LIN {X 0,Y 312.688,Z 380.055,A -85,B 0,C 180,E1 -15702.753,E2 -15702.753} C_VEL
LIN {X 0,Y 311.794,Z 385.413,A -85,B 0,C 180,E1 -15704.959,E2 -15704.959} C_VEL
LIN {X 0,Y 311.134,Z 389.57,A -85,B 0,C 180,E1 -15707.342,E2 -15707.342} C_VEL
LIN {X 0,Y 310.753,Z 391.625,A -85,B 0,C 180,E1 -15709.017,E2 -15709.017} C_VEL
LIN {X 0,Y 310.505,Z 392.931,A -85,B 0,C 180,E1 -15710.675,E2 -15710.675} C_VEL
LIN {X 0,Y 310.399,Z 393.625,A -85,B 0,C 180,E1 -15712.415,E2 -15712.415} C_VEL
LIN {X 0,Y 310.321,Z 393.447,A -85,B 0,C 180,E1 -15714.617,E2 -15714.617} C_VEL
LIN {X 0,Y 310.452,Z 391.861,A -85,B 0,C 180,E1 -15717.093,E2 -15717.093} C_VEL
LIN {X 0,Y 310.763,Z 389.249,A -85,B 0,C 180,E1 -15719.246,E2 -15719.246} C_VEL
LIN {X 0,Y 311.221,Z 384.676,A -85,B 0,C 180,E1 -15721.725,E2 -15721.725} C_VEL
LIN {X 0,Y 311.824,Z 379.437,A -85,B 0,C 180,E1 -15723.802,E2 -15723.802} C_VEL
LIN {X 0,Y 312.576,Z 373.086,A -85,B 0,C 180,E1 -15725.776,E2 -15725.776} C_VEL
LIN {X 0,Y 313.482,Z 365.782,A -85,B 0,C 180,E1 -15727.598,E2 -15727.598} C_VEL
LIN {X 0,Y 314.661,Z 356.752,A -85,B 0,C 180,E1 -15729.403,E2 -15729.403} C_VEL
LIN {X 0,Y 315.916,Z 346.753,A -85,B 0,C 180,E1 -15731.015,E2 -15731.015} C_VEL
LIN {X 0,Y 317.246,Z 335.532,A -85,B 0,C 180,E1 -15732.453,E2 -15732.453} C_VEL
LIN {X 0,Y 318.469,Z 323.461,A -85,B 0,C 180,E1 -15733.66,E2 -15733.66} C_VEL
LIN {X 0,Y 319.474,Z 310.963,A -85,B 0,C 180,E1 -15734.613,E2 -15734.613} C_VEL
LIN {X 0,Y 320.299,Z 298.124,A -85,B 0,C 180,E1 -15735.304,E2 -15735.304} C_VEL
LIN {X 0,Y 320.899,Z 284.464,A -85,B 0,C 180,E1 -15735.77,E2 -15735.77} C_VEL
LIN {X 0,Y 322.484,Z 214.178,A -85,B 0,C 180,E1 -15737.436,E2 -15737.436} C_VEL
LIN {X 0,Y 318.5,Z 192.839,A -85,B 0,C 180,E1 -15738.248,E2 -15738.248} C_VEL
LIN {X 0,Y 315.024,Z 182.877,A -85,B 0,C 180,E1 -15738.777,E2 -15738.777} C_VEL
LIN {X 0,Y 314.543,Z 180.395,A -85,B 0,C 180,E1 -15739.453,E2 -15739.453} C_VEL
LIN {X 0,Y 312.923,Z 171.315,A -85,B 0,C 180,E1 -15742.419,E2 -15742.419} C_VEL
LIN {X 0,Y 312.873,Z 171.01,A -85,B 0,C 180,E1 -15742.905,E2 -15742.905} C_VEL
LIN {X 0,Y 312.933,Z 171.005,A -85,B 0,C 180,E1 -15747.427,E2 -15747.427} C_VEL
LIN {X 0,Y 313.099,Z 170.983,A -85,B 0,C 180,E1 -15750.001,E2 -15750.001} C_VEL
LIN {X 0,Y 312.934,Z 171.002,A -85,B 0,C 180,E1 -15752.576,E2 -15752.576} C_VEL
LIN {X 0,Y 312.89,Z 171.008,A -85,B 0,C 180,E1 -15756.45,E2 -15756.45} C_VEL
LIN {X 0,Y 312.684,Z 171.033,A -85,B 0,C 180,E1 -15760.36,E2 -15760.36} C_VEL
LIN {X 0,Y 312.699,Z 171.032,A -85,B 0,C 180,E1 -15764.889,E2 -15764.889} C_VEL
LIN {X 0,Y 312.63,Z 171.041,A -85,B 0,C 180,E1 -15769.238,E2 -15769.238} C_VEL
LIN {X 0,Y 312.545,Z 171.052,A -85,B 0,C 180,E1 -15772.79,E2 -15772.79} C_VEL
LIN {X 0,Y 312.596,Z 171.039,A -85,B 0,C 180,E1 -15775.934,E2 -15775.934} C_VEL
LIN {X 0,Y 312.538,Z 171.052,A -85,B 0,C 180,E1 -15779.652,E2 -15779.652} C_VEL
LIN {X 0,Y 312.519,Z 171.052,A -85,B 0,C 180,E1 -15783.69,E2 -15783.69} C_VEL
LIN {X 0,Y 312.52,Z 171.051,A -85,B 0,C 180,E1 -15787.387,E2 -15787.387} C_VEL
LIN {X 0,Y 312.49,Z 171.06,A -85,B 0,C 180,E1 -15790.71,E2 -15790.71} C_VEL
LIN {X 0,Y 312.473,Z 171.059,A -85,B 0,C 180,E1 -15794.207,E2 -15794.207} C_VEL
LIN {X 0,Y 312.447,Z 171.057,A -85,B 0,C 180,E1 -15795.292,E2 -15795.292} C_VEL
LIN {X 0,Y 311.803,Z 171.141,A -85,B 0,C 180,E1 -15796.368,E2 -15796.368} C_VEL
LIN {X 0,Y 308.949,Z 171.49,A -85,B 0,C 180,E1 -15798.119,E2 -15798.119} C_VEL
LIN {X 0,Y 306.523,Z 171.792,A -85,B 0,C 180,E1 -15799.54,E2 -15799.54} C_VEL
LIN {X 0,Y 305.494,Z 171.926,A -85,B 0,C 180,E1 -15800.64,E2 -15800.64} C_VEL
LIN {X 0,Y 305.417,Z 171.93,A -85,B 0,C 180,E1 -15801.012,E2 -15801.012} C_VEL
LIN {X 0,Y 305.462,Z 171.935,A -85,B 0,C 180,E1 -15804.888,E2 -15804.888} C_VEL
LIN {X 0,Y 305.442,Z 171.938,A -85,B 0,C 180,E1 -15808.359,E2 -15808.359} C_VEL
LIN {X 0,Y 305.477,Z 171.931,A -85,B 0,C 180,E1 -15811.11,E2 -15811.11} C_VEL
LIN {X 0,Y 305.502,Z 171.93,A -85,B 0,C 180,E1 -15814.082,E2 -15814.082} C_VEL
LIN {X 0,Y 305.484,Z 171.933,A -85,B 0,C 180,E1 -15818.402,E2 -15818.402} C_VEL
LIN {X 0,Y 305.591,Z 171.916,A -85,B 0,C 180,E1 -15821.218,E2 -15821.218} C_VEL
LIN {X 0,Y 305.651,Z 171.906,A -85,B 0,C 180,E1 -15825.35,E2 -15825.35} C_VEL
LIN {X 0,Y 305.626,Z 171.913,A -85,B 0,C 180,E1 -15829.4,E2 -15829.4} C_VEL
LIN {X 0,Y 305.748,Z 171.898,A -85,B 0,C 180,E1 -15832.073,E2 -15832.073} C_VEL
LIN {X 0,Y 305.659,Z 171.908,A -85,B 0,C 180,E1 -15834.724,E2 -15834.724} C_VEL
LIN {X 0,Y 305.948,Z 171.87,A -85,B 0,C 180,E1 -15838.684,E2 -15838.684} C_VEL
LIN {X 0,Y 305.938,Z 171.87,A -85,B 0,C 180,E1 -15841.317,E2 -15841.317} C_VEL
LIN {X 0,Y 305.662,Z 171.902,A -85,B 0,C 180,E1 -15845.278,E2 -15845.278} C_VEL
LIN {X 0,Y 305.748,Z 171.899,A -85,B 0,C 180,E1 -15847.928,E2 -15847.928} C_VEL
LIN {X 0,Y 305.6,Z 171.916,A -85,B 0,C 180,E1 -15851.946,E2 -15851.946} C_VEL
LIN {X 0,Y 305.612,Z 171.91,A -85,B 0,C 180,E1 -15855.014,E2 -15855.014} C_VEL
LIN {X 0,Y 305.518,Z 171.924,A -85,B 0,C 180,E1 -15858.788,E2 -15858.788} C_VEL
LIN {X 0,Y 305.459,Z 171.936,A -85,B 0,C 180,E1 -15863.026,E2 -15863.026} C_VEL
LIN {X 0,Y 305.454,Z 171.928,A -85,B 0,C 180,E1 -15866.19,E2 -15866.19} C_VEL
LIN {X 0,Y 305.449,Z 171.937,A -85,B 0,C 180,E1 -15869.033,E2 -15869.033} C_VEL
LIN {X 0,Y 305.438,Z 171.935,A -85,B 0,C 180,E1 -15871.953,E2 -15871.953} C_VEL
LIN {X 0,Y 305.464,Z 171.934,A -85,B 0,C 180,E1 -15875.114,E2 -15875.114} C_VEL
LIN {X 0,Y 305.436,Z 171.938,A -85,B 0,C 180,E1 -15878.525,E2 -15878.525} C_VEL
LIN {X 0,Y 305.438,Z 171.939,A -85,B 0,C 180,E1 -15882.581,E2 -15882.581} C_VEL
LIN {X 0,Y 305.424,Z 171.938,A -85,B 0,C 180,E1 -15886.344,E2 -15886.344} C_VEL
LIN {X 0,Y 305.414,Z 171.94,A -85,B 0,C 180,E1 -15889.884,E2 -15889.884} C_VEL
LIN {X 0,Y 305.463,Z 171.934,A -85,B 0,C 180,E1 -15893.637,E2 -15893.637} C_VEL
LIN {X 0,Y 305.467,Z 171.936,A -85,B 0,C 180,E1 -15896.482,E2 -15896.482} C_VEL
LIN {X 0,Y 305.474,Z 172.085,A -85,B 0,C 180,E1 -15898.652,E2 -15898.652} C_VEL
LIN {X 0,Y 307.663,Z 182.551,A -85,B 0,C 180,E1 -15902.077,E2 -15902.077} C_VEL
LIN {X 0,Y 309.377,Z 191.56,A -85,B 0,C 180,E1 -15904.816,E2 -15904.816} C_VEL
LIN {X 0,Y 310.305,Z 195.562,A -85,B 0,C 180,E1 -15905.043,E2 -15905.043} C_VEL
LIN {X 0,Y 315.736,Z 229.812,A -85,B 0,C 180,E1 -15906.314,E2 -15906.314} C_VEL
LIN {X 0,Y 313.948,Z 299.456,A -85,B 0,C 180,E1 -15908.02,E2 -15908.02} C_VEL
LIN {X 0,Y 313.1,Z 313.167,A -85,B 0,C 180,E1 -15908.606,E2 -15908.606} C_VEL
LIN {X 0,Y 312.112,Z 325.64,A -85,B 0,C 180,E1 -15909.399,E2 -15909.399} C_VEL
LIN {X 0,Y 310.969,Z 336.814,A -85,B 0,C 180,E1 -15910.355,E2 -15910.355} C_VEL
LIN {X 0,Y 309.603,Z 348.458,A -85,B 0,C 180,E1 -15911.64,E2 -15911.64} C_VEL
LIN {X 0,Y 308.323,Z 359.263,A -85,B 0,C 180,E1 -15913.15,E2 -15913.15} C_VEL
LIN {X 0,Y 307.15,Z 368.404,A -85,B 0,C 180,E1 -15914.743,E2 -15914.743} C_VEL
LIN {X 0,Y 305.891,Z 377.519,A -85,B 0,C 180,E1 -15916.716,E2 -15916.716} C_VEL
LIN {X 0,Y 304.97,Z 384.854,A -85,B 0,C 180,E1 -15918.703,E2 -15918.703} C_VEL
LIN {X 0,Y 304.295,Z 390.695,A -85,B 0,C 180,E1 -15920.695,E2 -15920.695} C_VEL
LIN {X 0,Y 303.851,Z 395.272,A -85,B 0,C 180,E1 -15922.69,E2 -15922.69} C_VEL
LIN {X 0,Y 303.64,Z 398.735,A -85,B 0,C 180,E1 -15924.686,E2 -15924.686} C_VEL
LIN {X 0,Y 303.586,Z 400.449,A -85,B 0,C 180,E1 -15926.016,E2 -15926.016} C_VEL
LIN {X 0,Y 303.58,Z 401.75,A -85,B 0,C 180,E1 -15927.345,E2 -15927.345} C_VEL
LIN {X 0,Y 303.529,Z 402.647,A -85,B 0,C 180,E1 -15928.672,E2 -15928.672} C_VEL
LIN {X 0,Y 303.546,Z 403.111,A -85,B 0,C 180,E1 -15929.999,E2 -15929.999} C_VEL
LIN {X 0,Y 303.583,Z 402.812,A -85,B 0,C 180,E1 -15932.652,E2 -15932.652} C_VEL
LIN {X 0,Y 303.605,Z 402.078,A -85,B 0,C 180,E1 -15933.981,E2 -15933.981} C_VEL
LIN {X 0,Y 303.732,Z 400.43,A -85,B 0,C 180,E1 -15935.744,E2 -15935.744} C_VEL
LIN {X 0,Y 304.065,Z 397.307,A -85,B 0,C 180,E1 -15937.97,E2 -15937.97} C_VEL
LIN {X 0,Y 304.673,Z 393.415,A -85,B 0,C 180,E1 -15939.961,E2 -15939.961} C_VEL
LIN {X 0,Y 305.52,Z 388.396,A -85,B 0,C 180,E1 -15941.947,E2 -15941.947} C_VEL
LIN {X 0,Y 306.648,Z 382.103,A -85,B 0,C 180,E1 -15943.923,E2 -15943.923} C_VEL
LIN {X 0,Y 308.286,Z 374.24,A -85,B 0,C 180,E1 -15945.875,E2 -15945.875} C_VEL
LIN {X 0,Y 309.58,Z 366.049,A -85,B 0,C 180,E1 -15947.545,E2 -15947.545} C_VEL
LIN {X 0,Y 311.45,Z 355.494,A -85,B 0,C 180,E1 -15949.268,E2 -15949.268} C_VEL
LIN {X 0,Y 313.221,Z 344.43,A -85,B 0,C 180,E1 -15950.693,E2 -15950.693} C_VEL
LIN {X 0,Y 315.075,Z 331.897,A -85,B 0,C 180,E1 -15951.937,E2 -15951.937} C_VEL
LIN {X 0,Y 316.504,Z 319.535,A -85,B 0,C 180,E1 -15952.865,E2 -15952.865} C_VEL
LIN {X 0,Y 317.63,Z 306.569,A -85,B 0,C 180,E1 -15953.555,E2 -15953.555} C_VEL
LIN {X 0,Y 318.347,Z 293.048,A -85,B 0,C 180,E1 -15954.017,E2 -15954.017} C_VEL
LIN {X 0,Y 320.362,Z 231.537,A -85,B 0,C 180,E1 -15955.514,E2 -15955.514} C_VEL
LIN {X 0,Y 317.662,Z 214.971,A -85,B 0,C 180,E1 -15956.26,E2 -15956.26} C_VEL
LIN {X 0,Y 314.964,Z 202.486,A -85,B 0,C 180,E1 -15956.915,E2 -15956.915} C_VEL
LIN {X 0,Y 309.876,Z 190.776,A -85,B 0,C 180,E1 -15957.887,E2 -15957.887} C_VEL
LIN {X 0,Y 307.917,Z 181.754,A -85,B 0,C 180,E1 -15960.898,E2 -15960.898} C_VEL
LIN {X 0,Y 305.532,Z 172.315,A -85,B 0,C 180,E1 -15964.383,E2 -15964.383} C_VEL
LIN {X 0,Y 305.442,Z 171.957,A -85,B 0,C 180,E1 -15964.681,E2 -15964.681} C_VEL
LIN {X 0,Y 305.41,Z 171.941,A -85,B 0,C 180,E1 -15968.518,E2 -15968.518} C_VEL
LIN {X 0,Y 305.428,Z 171.94,A -85,B 0,C 180,E1 -15972.579,E2 -15972.579} C_VEL
LIN {X 0,Y 305.413,Z 171.94,A -85,B 0,C 180,E1 -15976.342,E2 -15976.342} C_VEL
LIN {X 0,Y 305.402,Z 171.94,A -85,B 0,C 180,E1 -15979.883,E2 -15979.883} C_VEL
LIN {X 0,Y 305.454,Z 171.938,A -85,B 0,C 180,E1 -15983.635,E2 -15983.635} C_VEL
LIN {X 0,Y 305.456,Z 171.932,A -85,B 0,C 180,E1 -15986.481,E2 -15986.481} C_VEL
LIN {X 0,Y 305.42,Z 171.934,A -85,B 0,C 180,E1 -15989.586,E2 -15989.586} C_VEL
LIN {X 0,Y 305.444,Z 171.93,A -85,B 0,C 180,E1 -15992.601,E2 -15992.601} C_VEL
LIN {X 0,Y 305.463,Z 171.932,A -85,B 0,C 180,E1 -15995.534,E2 -15995.534} C_VEL
LIN {X 0,Y 305.473,Z 171.929,A -85,B 0,C 180,E1 -15999.811,E2 -15999.811} C_VEL
LIN {X 0,Y 305.54,Z 171.92,A -85,B 0,C 180,E1 -16003.976,E2 -16003.976} C_VEL
LIN {X 0,Y 305.576,Z 171.922,A -85,B 0,C 180,E1 -16006.703,E2 -16006.703} C_VEL
LIN {X 0,Y 305.741,Z 171.899,A -85,B 0,C 180,E1 -16011.261,E2 -16011.261} C_VEL
LIN {X 0,Y 305.787,Z 171.889,A -85,B 0,C 180,E1 -16013.401,E2 -16013.401} C_VEL
LIN {X 0,Y 305.847,Z 171.883,A -85,B 0,C 180,E1 -16017.365,E2 -16017.365} C_VEL
LIN {X 0,Y 305.9,Z 171.873,A -85,B 0,C 180,E1 -16019.999,E2 -16019.999} C_VEL
LIN {X 0,Y 305.843,Z 171.884,A -85,B 0,C 180,E1 -16022.634,E2 -16022.634} C_VEL
LIN {X 0,Y 305.787,Z 171.891,A -85,B 0,C 180,E1 -16026.644,E2 -16026.644} C_VEL
LIN {X 0,Y 305.681,Z 171.904,A -85,B 0,C 180,E1 -16029.261,E2 -16029.261} C_VEL
LIN {X 0,Y 305.572,Z 171.922,A -85,B 0,C 180,E1 -16033.296,E2 -16033.296} C_VEL
LIN {X 0,Y 305.538,Z 171.925,A -85,B 0,C 180,E1 -16036.022,E2 -16036.022} C_VEL
LIN {X 0,Y 305.471,Z 171.937,A -85,B 0,C 180,E1 -16040.188,E2 -16040.188} C_VEL
LIN {X 0,Y 305.502,Z 172.159,A -85,B 0,C 180,E1 -16041.951,E2 -16041.951} C_VEL
LIN {X 0,Y 307.553,Z 180.233,A -85,B 0,C 180,E1 -16045.008,E2 -16045.008} C_VEL
LIN {X 0,Y 308.206,Z 183.045,A -85,B 0,C 180,E1 -16045.946,E2 -16045.946} C_VEL
LIN {X 0,Y 315.382,Z 198.321,A -85,B 0,C 180,E1 -16047.287,E2 -16047.287} C_VEL
LIN {X 0,Y 318.646,Z 206.73,A -85,B 0,C 180,E1 -16047.887,E2 -16047.887} C_VEL
LIN {X 0,Y 320.722,Z 217.922,A -85,B 0,C 180,E1 -16048.419,E2 -16048.419} C_VEL
LIN {X 0,Y 318.277,Z 291.184,A -85,B 0,C 180,E1 -16050.243,E2 -16050.243} C_VEL
LIN {X 0,Y 317.366,Z 304.177,A -85,B 0,C 180,E1 -16050.804,E2 -16050.804} C_VEL
LIN {X 0,Y 316.218,Z 316.908,A -85,B 0,C 180,E1 -16051.62,E2 -16051.62} C_VEL
LIN {X 0,Y 314.711,Z 329.185,A -85,B 0,C 180,E1 -16052.692,E2 -16052.692} C_VEL
LIN {X 0,Y 313.176,Z 339.725,A -85,B 0,C 180,E1 -16053.872,E2 -16053.872} C_VEL
LIN {X 0,Y 311.372,Z 350.484,A -85,B 0,C 180,E1 -16055.379,E2 -16055.379} C_VEL
LIN {X 0,Y 309.57,Z 360.286,A -85,B 0,C 180,E1 -16057.119,E2 -16057.119} C_VEL
LIN {X 0,Y 307.913,Z 369.208,A -85,B 0,C 180,E1 -16059.104,E2 -16059.104} C_VEL
LIN {X 0,Y 306.67,Z 375.582,A -85,B 0,C 180,E1 -16060.867,E2 -16060.867} C_VEL
LIN {X 0,Y 305.381,Z 382.238,A -85,B 0,C 180,E1 -16063.212,E2 -16063.212} C_VEL
LIN {X 0,Y 304.458,Z 387.472,A -85,B 0,C 180,E1 -16065.691,E2 -16065.691} C_VEL
LIN {X 0,Y 303.925,Z 390.724,A -85,B 0,C 180,E1 -16067.889,E2 -16067.889} C_VEL
LIN {X 0,Y 303.514,Z 392.608,A -85,B 0,C 180,E1 -16069.829,E2 -16069.829} C_VEL
LIN {X 0,Y 303.306,Z 393.682,A -85,B 0,C 180,E1 -16071.982,E2 -16071.982} C_VEL
LIN {X 0,Y 303.245,Z 393.542,A -85,B 0,C 180,E1 -16074.594,E2 -16074.594} C_VEL
LIN {X 0,Y 303.289,Z 392.451,A -85,B 0,C 180,E1 -16076.533,E2 -16076.533} C_VEL
LIN {X 0,Y 303.619,Z 389.865,A -85,B 0,C 180,E1 -16078.919,E2 -16078.919} C_VEL
LIN {X 0,Y 303.97,Z 386.545,A -85,B 0,C 180,E1 -16080.955,E2 -16080.955} C_VEL
LIN {X 0,Y 304.517,Z 381.431,A -85,B 0,C 180,E1 -16083.256,E2 -16083.256} C_VEL
LIN {X 0,Y 305.175,Z 375.94,A -85,B 0,C 180,E1 -16085.158,E2 -16085.158} C_VEL
LIN {X 0,Y 306.018,Z 369.268,A -85,B 0,C 180,E1 -16087.021,E2 -16087.021} C_VEL
LIN {X 0,Y 307.289,Z 360.041,A -85,B 0,C 180,E1 -16089.068,E2 -16089.068} C_VEL
LIN {X 0,Y 308.503,Z 350.822,A -85,B 0,C 180,E1 -16090.713,E2 -16090.713} C_VEL
LIN {X 0,Y 309.791,Z 340.925,A -85,B 0,C 180,E1 -16092.141,E2 -16092.141} C_VEL
LIN {X 0,Y 311.032,Z 329.763,A -85,B 0,C 180,E1 -16093.427,E2 -16093.427} C_VEL
LIN {X 0,Y 312.249,Z 317.351,A -85,B 0,C 180,E1 -16094.538,E2 -16094.538} C_VEL
LIN {X 0,Y 313.132,Z 304.949,A -85,B 0,C 180,E1 -16095.362,E2 -16095.362} C_VEL
LIN {X 0,Y 313.914,Z 291.826,A -85,B 0,C 180,E1 -16095.951,E2 -16095.951} C_VEL
LIN {X 0,Y 314.735,Z 261.534,A -85,B 0,C 180,E1 -16096.729,E2 -16096.729} C_VEL
LIN {X 0,Y 315.866,Z 215.349,A -85,B 0,C 180,E1 -16097.847,E2 -16097.847} C_VEL
LIN {X 0,Y 312.086,Z 195.088,A -85,B 0,C 180,E1 -16098.637,E2 -16098.637} C_VEL
LIN {X 0,Y 307.81,Z 182.861,A -85,B 0,C 180,E1 -16099.311,E2 -16099.311} C_VEL
LIN {X 0,Y 305.894,Z 172.261,A -85,B 0,C 180,E1 -16102.742,E2 -16102.742} C_VEL
LIN {X 0,Y 305.833,Z 171.887,A -85,B 0,C 180,E1 -16103.072,E2 -16103.072} C_VEL
LIN {X 0,Y 305.882,Z 171.883,A -85,B 0,C 180,E1 -16107.368,E2 -16107.368} C_VEL
LIN {X 0,Y 306.051,Z 171.861,A -85,B 0,C 180,E1 -16110.001,E2 -16110.001} C_VEL
LIN {X 0,Y 305.882,Z 171.881,A -85,B 0,C 180,E1 -16112.635,E2 -16112.635} C_VEL
LIN {X 0,Y 305.83,Z 171.887,A -85,B 0,C 180,E1 -16116.599,E2 -16116.599} C_VEL
LIN {X 0,Y 305.692,Z 171.905,A -85,B 0,C 180,E1 -16119.262,E2 -16119.262} C_VEL
LIN {X 0,Y 305.588,Z 171.918,A -85,B 0,C 180,E1 -16123.297,E2 -16123.297} C_VEL
LIN {X 0,Y 305.593,Z 171.917,A -85,B 0,C 180,E1 -16126.021,E2 -16126.021} C_VEL
LIN {X 0,Y 305.576,Z 171.919,A -85,B 0,C 180,E1 -16129.446,E2 -16129.446} C_VEL
LIN {X 0,Y 305.49,Z 171.933,A -85,B 0,C 180,E1 -16133.043,E2 -16133.043} C_VEL
LIN {X 0,Y 305.525,Z 171.919,A -85,B 0,C 180,E1 -16136.22,E2 -16136.22} C_VEL
LIN {X 0,Y 305.488,Z 171.932,A -85,B 0,C 180,E1 -16139.049,E2 -16139.049} C_VEL
LIN {X 0,Y 305.442,Z 171.935,A -85,B 0,C 180,E1 -16141.953,E2 -16141.953} C_VEL
LIN {X 0,Y 305.462,Z 171.929,A -85,B 0,C 180,E1 -16145.114,E2 -16145.114} C_VEL
LIN {X 0,Y 305.44,Z 171.933,A -85,B 0,C 180,E1 -16148.527,E2 -16148.527} C_VEL
LIN {X 0,Y 305.459,Z 171.936,A -85,B 0,C 180,E1 -16152.588,E2 -16152.588} C_VEL
LIN {X 0,Y 305.442,Z 171.933,A -85,B 0,C 180,E1 -16156.349,E2 -16156.349} C_VEL
LIN {X 0,Y 305.458,Z 171.925,A -85,B 0,C 180,E1 -16159.893,E2 -16159.893} C_VEL
LIN {X 0,Y 305.417,Z 171.93,A -85,B 0,C 180,E1 -16161.012,E2 -16161.012} C_VEL
LIN {X 0,Y 304.762,Z 172.019,A -85,B 0,C 180,E1 -16162.112,E2 -16162.112} C_VEL
LIN {X 0,Y 301.894,Z 172.377,A -85,B 0,C 180,E1 -16163.903,E2 -16163.903} C_VEL
LIN {X 0,Y 299.467,Z 172.68,A -85,B 0,C 180,E1 -16165.356,E2 -16165.356} C_VEL
LIN {X 0,Y 298.447,Z 172.811,A -85,B 0,C 180,E1 -16166.481,E2 -16166.481} C_VEL
LIN {X 0,Y 298.377,Z 172.812,A -85,B 0,C 180,E1 -16166.862,E2 -16166.862} C_VEL
LIN {X 0,Y 298.403,Z 172.815,A -85,B 0,C 180,E1 -16170.626,E2 -16170.626} C_VEL
LIN {X 0,Y 298.446,Z 172.806,A -85,B 0,C 180,E1 -16174.921,E2 -16174.921} C_VEL
LIN {X 0,Y 298.442,Z 172.806,A -85,B 0,C 180,E1 -16179.315,E2 -16179.315} C_VEL
LIN {X 0,Y 298.539,Z 172.798,A -85,B 0,C 180,E1 -16182.18,E2 -16182.18} C_VEL
LIN {X 0,Y 298.595,Z 172.784,A -85,B 0,C 180,E1 -16184.996,E2 -16184.996} C_VEL
LIN {X 0,Y 298.585,Z 172.789,A -85,B 0,C 180,E1 -16189.147,E2 -16189.147} C_VEL
LIN {X 0,Y 298.7,Z 172.776,A -85,B 0,C 180,E1 -16191.885,E2 -16191.885} C_VEL
LIN {X 0,Y 298.629,Z 172.784,A -85,B 0,C 180,E1 -16194.599,E2 -16194.599} C_VEL
LIN {X 0,Y 298.915,Z 172.746,A -85,B 0,C 180,E1 -16198.653,E2 -16198.653} C_VEL
LIN {X 0,Y 298.906,Z 172.745,A -85,B 0,C 180,E1 -16201.348,E2 -16201.348} C_VEL
LIN {X 0,Y 298.735,Z 172.767,A -85,B 0,C 180,E1 -16206.756,E2 -16206.756} C_VEL
LIN {X 0,Y 298.629,Z 172.788,A -85,B 0,C 180,E1 -16209.483,E2 -16209.483} C_VEL
LIN {X 0,Y 298.547,Z 172.792,A -85,B 0,C 180,E1 -16213.616,E2 -16213.616} C_VEL
LIN {X 0,Y 298.484,Z 172.793,A -85,B 0,C 180,E1 -16216.413,E2 -16216.413} C_VEL
LIN {X 0,Y 298.443,Z 172.81,A -85,B 0,C 180,E1 -16219.616,E2 -16219.616} C_VEL
LIN {X 0,Y 298.385,Z 172.813,A -85,B 0,C 180,E1 -16223.604,E2 -16223.604} C_VEL
LIN {X 0,Y 298.405,Z 172.805,A -85,B 0,C 180,E1 -16226.583,E2 -16226.583} C_VEL
LIN {X 0,Y 298.395,Z 172.815,A -85,B 0,C 180,E1 -16229.644,E2 -16229.644} C_VEL
LIN {X 0,Y 298.395,Z 172.815,A -85,B 0,C 180,E1 -16232.801,E2 -16232.801} C_VEL
LIN {X 0,Y 298.407,Z 172.811,A -85,B 0,C 180,E1 -16236.072,E2 -16236.072} C_VEL
LIN {X 0,Y 298.377,Z 172.812,A -85,B 0,C 180,E1 -16239.492,E2 -16239.492} C_VEL
LIN {X 0,Y 298.373,Z 172.818,A -85,B 0,C 180,E1 -16243.097,E2 -16243.097} C_VEL
LIN {X 0,Y 298.374,Z 172.82,A -85,B 0,C 180,E1 -16246.914,E2 -16246.914} C_VEL
LIN {X 0,Y 298.357,Z 172.82,A -85,B 0,C 180,E1 -16251.018,E2 -16251.018} C_VEL
LIN {X 0,Y 298.406,Z 172.813,A -85,B 0,C 180,E1 -16253.927,E2 -16253.927} C_VEL
LIN {X 0,Y 298.395,Z 172.817,A -85,B 0,C 180,E1 -16257.199,E2 -16257.199} C_VEL
LIN {X 0,Y 298.425,Z 172.896,A -85,B 0,C 180,E1 -16258.222,E2 -16258.222} C_VEL
LIN {X 0,Y 300.355,Z 182.055,A -85,B 0,C 180,E1 -16261.334,E2 -16261.334} C_VEL
LIN {X 0,Y 302.182,Z 191.553,A -85,B 0,C 180,E1 -16264.296,E2 -16264.296} C_VEL
LIN {X 0,Y 303.764,Z 196.973,A -85,B 0,C 180,E1 -16264.605,E2 -16264.605} C_VEL
LIN {X 0,Y 309.056,Z 230.443,A -85,B 0,C 180,E1 -16265.884,E2 -16265.884} C_VEL
LIN {X 0,Y 307.175,Z 300.255,A -85,B 0,C 180,E1 -16267.642,E2 -16267.642} C_VEL
LIN {X 0,Y 306.298,Z 313.667,A -85,B 0,C 180,E1 -16268.24,E2 -16268.24} C_VEL
LIN {X 0,Y 305.231,Z 326.467,A -85,B 0,C 180,E1 -16269.09,E2 -16269.09} C_VEL
LIN {X 0,Y 303.872,Z 339.009,A -85,B 0,C 180,E1 -16270.229,E2 -16270.229} C_VEL
LIN {X 0,Y 302.545,Z 350.243,A -85,B 0,C 180,E1 -16271.547,E2 -16271.547} C_VEL
LIN {X 0,Y 301.249,Z 360.337,A -85,B 0,C 180,E1 -16273.042,E2 -16273.042} C_VEL
LIN {X 0,Y 300.013,Z 369.495,A -85,B 0,C 180,E1 -16274.719,E2 -16274.719} C_VEL
LIN {X 0,Y 298.764,Z 378.413,A -85,B 0,C 180,E1 -16276.74,E2 -16276.74} C_VEL
LIN {X 0,Y 297.842,Z 385.521,A -85,B 0,C 180,E1 -16278.773,E2 -16278.773} C_VEL
LIN {X 0,Y 297.088,Z 392.008,A -85,B 0,C 180,E1 -16281.153,E2 -16281.153} C_VEL
LIN {X 0,Y 296.7,Z 396.256,A -85,B 0,C 180,E1 -16283.197,E2 -16283.197} C_VEL
LIN {X 0,Y 296.555,Z 398.498,A -85,B 0,C 180,E1 -16284.559,E2 -16284.559} C_VEL
LIN {X 0,Y 296.489,Z 400.242,A -85,B 0,C 180,E1 -16285.921,E2 -16285.921} C_VEL
LIN {X 0,Y 296.485,Z 401.565,A -85,B 0,C 180,E1 -16287.281,E2 -16287.281} C_VEL
LIN {X 0,Y 296.451,Z 402.484,A -85,B 0,C 180,E1 -16288.64,E2 -16288.64} C_VEL
LIN {X 0,Y 296.464,Z 402.989,A -85,B 0,C 180,E1 -16289.999,E2 -16289.999} C_VEL
LIN {X 0,Y 296.45,Z 403.055,A -85,B 0,C 180,E1 -16291.357,E2 -16291.357} C_VEL
LIN {X 0,Y 296.488,Z 402.73,A -85,B 0,C 180,E1 -16292.716,E2 -16292.716} C_VEL
LIN {X 0,Y 296.509,Z 402.015,A -85,B 0,C 180,E1 -16294.076,E2 -16294.076} C_VEL
LIN {X 0,Y 296.632,Z 400.633,A -85,B 0,C 180,E1 -16295.674,E2 -16295.674} C_VEL
LIN {X 0,Y 297.033,Z 397.325,A -85,B 0,C 180,E1 -16298.16,E2 -16298.16} C_VEL
LIN {X 0,Y 297.648,Z 393.474,A -85,B 0,C 180,E1 -16300.199,E2 -16300.199} C_VEL
LIN {X 0,Y 298.54,Z 388.508,A -85,B 0,C 180,E1 -16302.23,E2 -16302.23} C_VEL
LIN {X 0,Y 299.77,Z 382.28,A -85,B 0,C 180,E1 -16304.249,E2 -16304.249} C_VEL
LIN {X 0,Y 301.468,Z 374.531,A -85,B 0,C 180,E1 -16306.244,E2 -16306.244} C_VEL
LIN {X 0,Y 302.767,Z 366.82,A -85,B 0,C 180,E1 -16307.876,E2 -16307.876} C_VEL
LIN {X 0,Y 304.567,Z 357.033,A -85,B 0,C 180,E1 -16309.546,E2 -16309.546} C_VEL
LIN {X 0,Y 306.454,Z 346.4,A -85,B 0,C 180,E1 -16310.996,E2 -16310.996} C_VEL
LIN {X 0,Y 308.01,Z 336.17,A -85,B 0,C 180,E1 -16312.114,E2 -16312.114} C_VEL
LIN {X 0,Y 309.651,Z 324.035,A -85,B 0,C 180,E1 -16313.135,E2 -16313.135} C_VEL
LIN {X 0,Y 311.026,Z 310.733,A -85,B 0,C 180,E1 -16313.954,E2 -16313.954} C_VEL
LIN {X 0,Y 311.916,Z 297.376,A -85,B 0,C 180,E1 -16314.5,E2 -16314.5} C_VEL
LIN {X 0,Y 314.138,Z 231.868,A -85,B 0,C 180,E1 -16316.156,E2 -16316.156} C_VEL
LIN {X 0,Y 311.103,Z 213.804,A -85,B 0,C 180,E1 -16317.021,E2 -16317.021} C_VEL
LIN {X 0,Y 309.166,Z 205.169,A -85,B 0,C 180,E1 -16317.499,E2 -16317.499} C_VEL
LIN {X 0,Y 304.422,Z 194.409,A -85,B 0,C 180,E1 -16318.41,E2 -16318.41} C_VEL
LIN {X 0,Y 302.636,Z 190.429,A -85,B 0,C 180,E1 -16318.817,E2 -16318.817} C_VEL
LIN {X 0,Y 300.801,Z 182.167,A -85,B 0,C 180,E1 -16321.713,E2 -16321.713} C_VEL
LIN {X 0,Y 298.448,Z 173.11,A -85,B 0,C 180,E1 -16325.232,E2 -16325.232} C_VEL
LIN {X 0,Y 298.399,Z 172.817,A -85,B 0,C 180,E1 -16326.07,E2 -16326.07} C_VEL
LIN {X 0,Y 298.343,Z 172.822,A -85,B 0,C 180,E1 -16329.494,E2 -16329.494} C_VEL
LIN {X 0,Y 298.364,Z 172.823,A -85,B 0,C 180,E1 -16333.095,E2 -16333.095} C_VEL
LIN {X 0,Y 298.363,Z 172.817,A -85,B 0,C 180,E1 -16336.913,E2 -16336.913} C_VEL
LIN {X 0,Y 298.377,Z 172.82,A -85,B 0,C 180,E1 -16341.009,E2 -16341.009} C_VEL
LIN {X 0,Y 298.396,Z 172.816,A -85,B 0,C 180,E1 -16343.926,E2 -16343.926} C_VEL
LIN {X 0,Y 298.384,Z 172.819,A -85,B 0,C 180,E1 -16347.198,E2 -16347.198} C_VEL
LIN {X 0,Y 298.392,Z 172.815,A -85,B 0,C 180,E1 -16350.624,E2 -16350.624} C_VEL
LIN {X 0,Y 298.428,Z 172.814,A -85,B 0,C 180,E1 -16354.918,E2 -16354.918} C_VEL
LIN {X 0,Y 298.391,Z 172.813,A -85,B 0,C 180,E1 -16357.861,E2 -16357.861} C_VEL
LIN {X 0,Y 298.454,Z 172.798,A -85,B 0,C 180,E1 -16360.75,E2 -16360.75} C_VEL
LIN {X 0,Y 298.575,Z 172.783,A -85,B 0,C 180,E1 -16364.993,E2 -16364.993} C_VEL
LIN {X 0,Y 298.571,Z 172.785,A -85,B 0,C 180,E1 -16369.145,E2 -16369.145} C_VEL
LIN {X 0,Y 298.698,Z 172.774,A -85,B 0,C 180,E1 -16371.884,E2 -16371.884} C_VEL
LIN {X 0,Y 298.625,Z 172.788,A -85,B 0,C 180,E1 -16374.598,E2 -16374.598} C_VEL
LIN {X 0,Y 298.891,Z 172.753,A -85,B 0,C 180,E1 -16378.652,E2 -16378.652} C_VEL
LIN {X 0,Y 298.902,Z 172.752,A -85,B 0,C 180,E1 -16381.347,E2 -16381.347} C_VEL
LIN {X 0,Y 298.74,Z 172.769,A -85,B 0,C 180,E1 -16386.755,E2 -16386.755} C_VEL
LIN {X 0,Y 298.612,Z 172.785,A -85,B 0,C 180,E1 -16389.482,E2 -16389.482} C_VEL
LIN {X 0,Y 298.532,Z 172.797,A -85,B 0,C 180,E1 -16393.616,E2 -16393.616} C_VEL
LIN {X 0,Y 298.471,Z 172.806,A -85,B 0,C 180,E1 -16396.412,E2 -16396.412} C_VEL
LIN {X 0,Y 298.433,Z 172.811,A -85,B 0,C 180,E1 -16399.619,E2 -16399.619} C_VEL
LIN {X 0,Y 298.431,Z 172.996,A -85,B 0,C 180,E1 -16401.137,E2 -16401.137} C_VEL
LIN {X 0,Y 300.452,Z 180.704,A -85,B 0,C 180,E1 -16404.185,E2 -16404.185} C_VEL
LIN {X 0,Y 301.097,Z 183.33,A -85,B 0,C 180,E1 -16405.073,E2 -16405.073} C_VEL
LIN {X 0,Y 308.839,Z 199.482,A -85,B 0,C 180,E1 -16406.57,E2 -16406.57} C_VEL
LIN {X 0,Y 312.731,Z 208.891,A -85,B 0,C 180,E1 -16407.295,E2 -16407.295} C_VEL
LIN {X 0,Y 314.583,Z 219.062,A -85,B 0,C 180,E1 -16407.798,E2 -16407.798} C_VEL
LIN {X 0,Y 312.036,Z 290.936,A -85,B 0,C 180,E1 -16409.625,E2 -16409.625} C_VEL
LIN {X 0,Y 311.04,Z 304.523,A -85,B 0,C 180,E1 -16410.221,E2 -16410.221} C_VEL
LIN {X 0,Y 309.865,Z 316.954,A -85,B 0,C 180,E1 -16411.033,E2 -16411.033} C_VEL
LIN {X 0,Y 308.37,Z 328.683,A -85,B 0,C 180,E1 -16412.065,E2 -16412.065} C_VEL
LIN {X 0,Y 306.617,Z 340.191,A -85,B 0,C 180,E1 -16413.374,E2 -16413.374} C_VEL
LIN {X 0,Y 304.924,Z 349.938,A -85,B 0,C 180,E1 -16414.762,E2 -16414.762} C_VEL
LIN {X 0,Y 303.275,Z 358.422,A -85,B 0,C 180,E1 -16416.24,E2 -16416.24} C_VEL
LIN {X 0,Y 301.6,Z 366.921,A -85,B 0,C 180,E1 -16418.069,E2 -16418.069} C_VEL
LIN {X 0,Y 300.204,Z 373.869,A -85,B 0,C 180,E1 -16419.918,E2 -16419.918} C_VEL
LIN {X 0,Y 298.782,Z 380.658,A -85,B 0,C 180,E1 -16422.192,E2 -16422.192} C_VEL
LIN {X 0,Y 297.967,Z 384.881,A -85,B 0,C 180,E1 -16423.999,E2 -16423.999} C_VEL
LIN {X 0,Y 297.3,Z 388.384,A -85,B 0,C 180,E1 -16425.902,E2 -16425.902} C_VEL
LIN {X 0,Y 296.677,Z 391.685,A -85,B 0,C 180,E1 -16428.451,E2 -16428.451} C_VEL
LIN {X 0,Y 296.361,Z 393.068,A -85,B 0,C 180,E1 -16430.189,E2 -16430.189} C_VEL
LIN {X 0,Y 296.225,Z 393.815,A -85,B 0,C 180,E1 -16431.916,E2 -16431.916} C_VEL
LIN {X 0,Y 296.144,Z 393.845,A -85,B 0,C 180,E1 -16433.791,E2 -16433.791} C_VEL
LIN {X 0,Y 296.166,Z 392.827,A -85,B 0,C 180,E1 -16436.154,E2 -16436.154} C_VEL
LIN {X 0,Y 296.467,Z 390.465,A -85,B 0,C 180,E1 -16438.583,E2 -16438.583} C_VEL
LIN {X 0,Y 296.91,Z 386.455,A -85,B 0,C 180,E1 -16441.139,E2 -16441.139} C_VEL
LIN {X 0,Y 297.445,Z 381.682,A -85,B 0,C 180,E1 -16443.327,E2 -16443.327} C_VEL
LIN {X 0,Y 298.3,Z 375.006,A -85,B 0,C 180,E1 -16445.652,E2 -16445.652} C_VEL
LIN {X 0,Y 299.188,Z 368.064,A -85,B 0,C 180,E1 -16447.562,E2 -16447.562} C_VEL
LIN {X 0,Y 300.429,Z 359.511,A -85,B 0,C 180,E1 -16449.46,E2 -16449.46} C_VEL
LIN {X 0,Y 301.683,Z 350.247,A -85,B 0,C 180,E1 -16451.126,E2 -16451.126} C_VEL
LIN {X 0,Y 303.078,Z 339.774,A -85,B 0,C 180,E1 -16452.631,E2 -16452.631} C_VEL
LIN {X 0,Y 304.36,Z 328.592,A -85,B 0,C 180,E1 -16453.915,E2 -16453.915} C_VEL
LIN {X 0,Y 305.548,Z 316.107,A -85,B 0,C 180,E1 -16455.026,E2 -16455.026} C_VEL
LIN {X 0,Y 306.531,Z 302.798,A -85,B 0,C 180,E1 -16455.881,E2 -16455.881} C_VEL
LIN {X 0,Y 307.318,Z 289.576,A -85,B 0,C 180,E1 -16456.445,E2 -16456.445} C_VEL
LIN {X 0,Y 309.12,Z 215.782,A -85,B 0,C 180,E1 -16458.298,E2 -16458.298} C_VEL
LIN {X 0,Y 305.72,Z 197.393,A -85,B 0,C 180,E1 -16459.038,E2 -16459.038} C_VEL
LIN {X 0,Y 300.591,Z 182.864,A -85,B 0,C 180,E1 -16459.86,E2 -16459.86} C_VEL
LIN {X 0,Y 298.834,Z 173.045,A -85,B 0,C 180,E1 -16463.164,E2 -16463.164} C_VEL
LIN {X 0,Y 298.731,Z 172.776,A -85,B 0,C 180,E1 -16463.924,E2 -16463.924} C_VEL
LIN {X 0,Y 298.921,Z 172.748,A -85,B 0,C 180,E1 -16468.654,E2 -16468.654} C_VEL
LIN {X 0,Y 298.92,Z 172.748,A -85,B 0,C 180,E1 -16471.349,E2 -16471.349} C_VEL
LIN {X 0,Y 298.774,Z 172.766,A -85,B 0,C 180,E1 -16476.756,E2 -16476.756} C_VEL
LIN {X 0,Y 298.624,Z 172.787,A -85,B 0,C 180,E1 -16479.484,E2 -16479.484} C_VEL
LIN {X 0,Y 298.551,Z 172.796,A -85,B 0,C 180,E1 -16483.617,E2 -16483.617} C_VEL
LIN {X 0,Y 298.548,Z 172.794,A -85,B 0,C 180,E1 -16486.41,E2 -16486.41} C_VEL
LIN {X 0,Y 298.511,Z 172.799,A -85,B 0,C 180,E1 -16489.656,E2 -16489.656} C_VEL
LIN {X 0,Y 298.457,Z 172.806,A -85,B 0,C 180,E1 -16493.599,E2 -16493.599} C_VEL
LIN {X 0,Y 298.485,Z 172.796,A -85,B 0,C 180,E1 -16496.576,E2 -16496.576} C_VEL
LIN {X 0,Y 298.416,Z 172.811,A -85,B 0,C 180,E1 -16499.643,E2 -16499.643} C_VEL
LIN {X 0,Y 298.395,Z 172.816,A -85,B 0,C 180,E1 -16502.801,E2 -16502.801} C_VEL
LIN {X 0,Y 298.444,Z 172.801,A -85,B 0,C 180,E1 -16506.808,E2 -16506.808} C_VEL
LIN {X 0,Y 298.388,Z 172.817,A -85,B 0,C 180,E1 -16511.089,E2 -16511.089} C_VEL
LIN {X 0,Y 298.389,Z 172.812,A -85,B 0,C 180,E1 -16515.042,E2 -16515.042} C_VEL
LIN {X 0,Y 298.387,Z 172.806,A -85,B 0,C 180,E1 -16518.914,E2 -16518.914} C_VEL
LIN {X 0,Y 298.429,Z 172.809,A -85,B 0,C 180,E1 -16523.198,E2 -16523.198} C_VEL
LIN {X 0,Y 298.377,Z 172.812,A -85,B 0,C 180,E1 -16526.862,E2 -16526.862} C_VEL
LIN {X 0,Y 297.745,Z 172.896,A -85,B 0,C 180,E1 -16527.989,E2 -16527.989} C_VEL
LIN {X 0,Y 294.912,Z 173.255,A -85,B 0,C 180,E1 -16529.825,E2 -16529.825} C_VEL
LIN {X 0,Y 292.486,Z 173.557,A -85,B 0,C 180,E1 -16531.314,E2 -16531.314} C_VEL
LIN {X 0,Y 291.439,Z 173.684,A -85,B 0,C 180,E1 -16532.468,E2 -16532.468} C_VEL
LIN {X 0,Y 291.352,Z 173.692,A -85,B 0,C 180,E1 -16532.859,E2 -16532.859} C_VEL
LIN {X 0,Y 291.374,Z 173.683,A -85,B 0,C 180,E1 -16537.3,E2 -16537.3} C_VEL
LIN {X 0,Y 291.46,Z 173.681,A -85,B 0,C 180,E1 -16540.271,E2 -16540.271} C_VEL
LIN {X 0,Y 291.543,Z 173.664,A -85,B 0,C 180,E1 -16544.635,E2 -16544.635} C_VEL
LIN {X 0,Y 291.531,Z 173.668,A -85,B 0,C 180,E1 -16548.881,E2 -16548.881} C_VEL
LIN {X 0,Y 291.653,Z 173.653,A -85,B 0,C 180,E1 -16551.688,E2 -16551.688} C_VEL
LIN {X 0,Y 291.599,Z 173.66,A -85,B 0,C 180,E1 -16554.468,E2 -16554.468} C_VEL
LIN {X 0,Y 291.881,Z 173.622,A -85,B 0,C 180,E1 -16558.621,E2 -16558.621} C_VEL
LIN {X 0,Y 291.873,Z 173.621,A -85,B 0,C 180,E1 -16561.38,E2 -16561.38} C_VEL
LIN {X 0,Y 291.687,Z 173.645,A -85,B 0,C 180,E1 -16566.92,E2 -16566.92} C_VEL
LIN {X 0,Y 291.571,Z 173.667,A -85,B 0,C 180,E1 -16569.714,E2 -16569.714} C_VEL
LIN {X 0,Y 291.518,Z 173.664,A -85,B 0,C 180,E1 -16573.951,E2 -16573.951} C_VEL
LIN {X 0,Y 291.429,Z 173.672,A -85,B 0,C 180,E1 -16576.822,E2 -16576.822} C_VEL
LIN {X 0,Y 291.395,Z 173.686,A -85,B 0,C 180,E1 -16579.842,E2 -16579.842} C_VEL
LIN {X 0,Y 291.329,Z 173.69,A -85,B 0,C 180,E1 -16584.212,E2 -16584.212} C_VEL
LIN {X 0,Y 291.353,Z 173.689,A -85,B 0,C 180,E1 -16587.279,E2 -16587.279} C_VEL
LIN {X 0,Y 291.32,Z 173.695,A -85,B 0,C 180,E1 -16590.439,E2 -16590.439} C_VEL
LIN {X 0,Y 291.346,Z 173.686,A -85,B 0,C 180,E1 -16593.699,E2 -16593.699} C_VEL
LIN {X 0,Y 291.362,Z 173.692,A -85,B 0,C 180,E1 -16597.249,E2 -16597.249} C_VEL
LIN {X 0,Y 291.304,Z 173.694,A -85,B 0,C 180,E1 -16600.648,E2 -16600.648} C_VEL
LIN {X 0,Y 291.286,Z 173.7,A -85,B 0,C 180,E1 -16604.404,E2 -16604.404} C_VEL
LIN {X 0,Y 291.299,Z 173.7,A -85,B 0,C 180,E1 -16608.411,E2 -16608.411} C_VEL
LIN {X 0,Y 291.388,Z 173.688,A -85,B 0,C 180,E1 -16612.916,E2 -16612.916} C_VEL
LIN {X 0,Y 291.346,Z 173.695,A -85,B 0,C 180,E1 -16616.301,E2 -16616.301} C_VEL
LIN {X 0,Y 291.372,Z 173.797,A -85,B 0,C 180,E1 -16617.837,E2 -16617.837} C_VEL
LIN {X 0,Y 293.296,Z 182.801,A -85,B 0,C 180,E1 -16620.971,E2 -16620.971} C_VEL
LIN {X 0,Y 294.972,Z 191.33,A -85,B 0,C 180,E1 -16623.717,E2 -16623.717} C_VEL
LIN {X 0,Y 297.248,Z 198.493,A -85,B 0,C 180,E1 -16624.15,E2 -16624.15} C_VEL
LIN {X 0,Y 302.38,Z 231.379,A -85,B 0,C 180,E1 -16625.441,E2 -16625.441} C_VEL
LIN {X 0,Y 300.475,Z 299.953,A -85,B 0,C 180,E1 -16627.207,E2 -16627.207} C_VEL
LIN {X 0,Y 299.578,Z 313.418,A -85,B 0,C 180,E1 -16627.817,E2 -16627.817} C_VEL
LIN {X 0,Y 298.478,Z 326.264,A -85,B 0,C 180,E1 -16628.684,E2 -16628.684} C_VEL
LIN {X 0,Y 297.142,Z 338.026,A -85,B 0,C 180,E1 -16629.761,E2 -16629.761} C_VEL
LIN {X 0,Y 295.72,Z 349.415,A -85,B 0,C 180,E1 -16631.105,E2 -16631.105} C_VEL
LIN {X 0,Y 294.485,Z 358.894,A -85,B 0,C 180,E1 -16632.504,E2 -16632.504} C_VEL
LIN {X 0,Y 293.423,Z 367.26,A -85,B 0,C 180,E1 -16634.01,E2 -16634.01} C_VEL
LIN {X 0,Y 292.262,Z 375.179,A -85,B 0,C 180,E1 -16635.729,E2 -16635.729} C_VEL
LIN {X 0,Y 291.066,Z 382.887,A -85,B 0,C 180,E1 -16637.802,E2 -16637.802} C_VEL
LIN {X 0,Y 290.438,Z 388.162,A -85,B 0,C 180,E1 -16639.542,E2 -16639.542} C_VEL
LIN {X 0,Y 289.882,Z 393.251,A -85,B 0,C 180,E1 -16641.634,E2 -16641.634} C_VEL
LIN {X 0,Y 289.532,Z 397.171,A -85,B 0,C 180,E1 -16643.728,E2 -16643.728} C_VEL
LIN {X 0,Y 289.396,Z 400.036,A -85,B 0,C 180,E1 -16645.821,E2 -16645.821} C_VEL
LIN {X 0,Y 289.393,Z 401.381,A -85,B 0,C 180,E1 -16647.215,E2 -16647.215} C_VEL
LIN {X 0,Y 289.374,Z 402.321,A -85,B 0,C 180,E1 -16648.607,E2 -16648.607} C_VEL
LIN {X 0,Y 289.384,Z 402.86,A -85,B 0,C 180,E1 -16649.999,E2 -16649.999} C_VEL
LIN {X 0,Y 289.374,Z 402.954,A -85,B 0,C 180,E1 -16651.39,E2 -16651.39} C_VEL
LIN {X 0,Y 289.396,Z 402.649,A -85,B 0,C 180,E1 -16652.782,E2 -16652.782} C_VEL
LIN {X 0,Y 289.417,Z 401.953,A -85,B 0,C 180,E1 -16654.176,E2 -16654.176} C_VEL
LIN {X 0,Y 289.518,Z 400.863,A -85,B 0,C 180,E1 -16655.571,E2 -16655.571} C_VEL
LIN {X 0,Y 289.711,Z 399.32,A -85,B 0,C 180,E1 -16656.965,E2 -16656.965} C_VEL
LIN {X 0,Y 290.19,Z 396.221,A -85,B 0,C 180,E1 -16659.056,E2 -16659.056} C_VEL
LIN {X 0,Y 290.901,Z 392.069,A -85,B 0,C 180,E1 -16661.142,E2 -16661.142} C_VEL
LIN {X 0,Y 292.153,Z 385.737,A -85,B 0,C 180,E1 -16663.563,E2 -16663.563} C_VEL
LIN {X 0,Y 293.732,Z 378.855,A -85,B 0,C 180,E1 -16665.613,E2 -16665.613} C_VEL
LIN {X 0,Y 295.296,Z 371.128,A -85,B 0,C 180,E1 -16667.478,E2 -16667.478} C_VEL
LIN {X 0,Y 297.129,Z 361.529,A -85,B 0,C 180,E1 -16669.336,E2 -16669.336} C_VEL
LIN {X 0,Y 299.223,Z 350.764,A -85,B 0,C 180,E1 -16670.987,E2 -16670.987} C_VEL
LIN {X 0,Y 301.062,Z 340.065,A -85,B 0,C 180,E1 -16672.291,E2 -16672.291} C_VEL
LIN {X 0,Y 302.794,Z 328.161,A -85,B 0,C 180,E1 -16673.419,E2 -16673.419} C_VEL
LIN {X 0,Y 304.275,Z 315.884,A -85,B 0,C 180,E1 -16674.292,E2 -16674.292} C_VEL
LIN {X 0,Y 305.408,Z 303.343,A -85,B 0,C 180,E1 -16674.921,E2 -16674.921} C_VEL
LIN {X 0,Y 306.091,Z 289.201,A -85,B 0,C 180,E1 -16675.361,E2 -16675.361} C_VEL
LIN {X 0,Y 308.047,Z 232.975,A -85,B 0,C 180,E1 -16676.8,E2 -16676.8} C_VEL
LIN {X 0,Y 305.208,Z 215.868,A -85,B 0,C 180,E1 -16677.645,E2 -16677.645} C_VEL
LIN {X 0,Y 303.489,Z 208.046,A -85,B 0,C 180,E1 -16678.096,E2 -16678.096} C_VEL
LIN {X 0,Y 298.552,Z 197.081,A -85,B 0,C 180,E1 -16679.077,E2 -16679.077} C_VEL
LIN {X 0,Y 295.478,Z 190.343,A -85,B 0,C 180,E1 -16679.757,E2 -16679.757} C_VEL
LIN {X 0,Y 293.392,Z 181.472,A -85,B 0,C 180,E1 -16683.027,E2 -16683.027} C_VEL
LIN {X 0,Y 291.386,Z 173.79,A -85,B 0,C 180,E1 -16686.22,E2 -16686.22} C_VEL
LIN {X 0,Y 291.289,Z 173.701,A -85,B 0,C 180,E1 -16690.647,E2 -16690.647} C_VEL
LIN {X 0,Y 291.275,Z 173.7,A -85,B 0,C 180,E1 -16694.402,E2 -16694.402} C_VEL
LIN {X 0,Y 291.287,Z 173.703,A -85,B 0,C 180,E1 -16698.41,E2 -16698.41} C_VEL
LIN {X 0,Y 291.326,Z 173.697,A -85,B 0,C 180,E1 -16701.153,E2 -16701.153} C_VEL
LIN {X 0,Y 291.347,Z 173.692,A -85,B 0,C 180,E1 -16704.623,E2 -16704.623} C_VEL
LIN {X 0,Y 291.357,Z 173.69,A -85,B 0,C 180,E1 -16707.948,E2 -16707.948} C_VEL
LIN {X 0,Y 291.334,Z 173.696,A -85,B 0,C 180,E1 -16711.152,E2 -16711.152} C_VEL
LIN {X 0,Y 291.348,Z 173.692,A -85,B 0,C 180,E1 -16714.265,E2 -16714.265} C_VEL
LIN {X 0,Y 291.354,Z 173.684,A -85,B 0,C 180,E1 -16717.297,E2 -16717.297} C_VEL
LIN {X 0,Y 291.382,Z 173.68,A -85,B 0,C 180,E1 -16720.264,E2 -16720.264} C_VEL
LIN {X 0,Y 291.487,Z 173.666,A -85,B 0,C 180,E1 -16724.664,E2 -16724.664} C_VEL
LIN {X 0,Y 291.518,Z 173.663,A -85,B 0,C 180,E1 -16728.879,E2 -16728.879} C_VEL
LIN {X 0,Y 291.65,Z 173.654,A -85,B 0,C 180,E1 -16731.686,E2 -16731.686} C_VEL
LIN {X 0,Y 291.595,Z 173.662,A -85,B 0,C 180,E1 -16734.467,E2 -16734.467} C_VEL
LIN {X 0,Y 291.859,Z 173.63,A -85,B 0,C 180,E1 -16738.62,E2 -16738.62} C_VEL
LIN {X 0,Y 291.868,Z 173.629,A -85,B 0,C 180,E1 -16741.379,E2 -16741.379} C_VEL
LIN {X 0,Y 291.691,Z 173.647,A -85,B 0,C 180,E1 -16746.919,E2 -16746.919} C_VEL
LIN {X 0,Y 291.555,Z 173.665,A -85,B 0,C 180,E1 -16749.714,E2 -16749.714} C_VEL
LIN {X 0,Y 291.502,Z 173.672,A -85,B 0,C 180,E1 -16753.951,E2 -16753.951} C_VEL
LIN {X 0,Y 291.416,Z 173.688,A -85,B 0,C 180,E1 -16756.821,E2 -16756.821} C_VEL
LIN {X 0,Y 291.398,Z 173.819,A -85,B 0,C 180,E1 -16760.229,E2 -16760.229} C_VEL
LIN {X 0,Y 293.684,Z 182.486,A -85,B 0,C 180,E1 -16763.817,E2 -16763.817} C_VEL
LIN {X 0,Y 294.024,Z 183.749,A -85,B 0,C 180,E1 -16764.14,E2 -16764.14} C_VEL
LIN {X 0,Y 301.175,Z 198.009,A -85,B 0,C 180,E1 -16765.575,E2 -16765.575} C_VEL
LIN {X 0,Y 306.857,Z 211.195,A -85,B 0,C 180,E1 -16766.686,E2 -16766.686} C_VEL
LIN {X 0,Y 308.507,Z 220.273,A -85,B 0,C 180,E1 -16767.15,E2 -16767.15} C_VEL
LIN {X 0,Y 305.84,Z 291.218,A -85,B 0,C 180,E1 -16768.988,E2 -16768.988} C_VEL
LIN {X 0,Y 304.826,Z 304.332,A -85,B 0,C 180,E1 -16769.572,E2 -16769.572} C_VEL
LIN {X 0,Y 303.531,Z 317.404,A -85,B 0,C 180,E1 -16770.444,E2 -16770.444} C_VEL
LIN {X 0,Y 301.921,Z 329.236,A -85,B 0,C 180,E1 -16771.516,E2 -16771.516} C_VEL
LIN {X 0,Y 300.095,Z 340.62,A -85,B 0,C 180,E1 -16772.847,E2 -16772.847} C_VEL
LIN {X 0,Y 298.111,Z 351.469,A -85,B 0,C 180,E1 -16774.457,E2 -16774.457} C_VEL
LIN {X 0,Y 296.175,Z 360.919,A -85,B 0,C 180,E1 -16776.22,E2 -16776.22} C_VEL
LIN {X 0,Y 294.242,Z 370.146,A -85,B 0,C 180,E1 -16778.389,E2 -16778.389} C_VEL
LIN {X 0,Y 292.749,Z 376.89,A -85,B 0,C 180,E1 -16780.404,E2 -16780.404} C_VEL
LIN {X 0,Y 291.543,Z 382.353,A -85,B 0,C 180,E1 -16782.451,E2 -16782.451} C_VEL
LIN {X 0,Y 290.683,Z 386.662,A -85,B 0,C 180,E1 -16784.518,E2 -16784.518} C_VEL
LIN {X 0,Y 289.859,Z 390.757,A -85,B 0,C 180,E1 -16787.245,E2 -16787.245} C_VEL
LIN {X 0,Y 289.48,Z 392.514,A -85,B 0,C 180,E1 -16789.045,E2 -16789.045} C_VEL
LIN {X 0,Y 289.188,Z 393.688,A -85,B 0,C 180,E1 -16791.048,E2 -16791.048} C_VEL
LIN {X 0,Y 289.056,Z 394.001,A -85,B 0,C 180,E1 -16793.354,E2 -16793.354} C_VEL
LIN {X 0,Y 289.06,Z 393.007,A -85,B 0,C 180,E1 -16796.001,E2 -16796.001} C_VEL
LIN {X 0,Y 289.314,Z 391.01,A -85,B 0,C 180,E1 -16798.234,E2 -16798.234} C_VEL
LIN {X 0,Y 289.742,Z 387.271,A -85,B 0,C 180,E1 -16800.833,E2 -16800.833} C_VEL
LIN {X 0,Y 290.3,Z 382.571,A -85,B 0,C 180,E1 -16803.131,E2 -16803.131} C_VEL
LIN {X 0,Y 291.056,Z 376.536,A -85,B 0,C 180,E1 -16805.386,E2 -16805.386} C_VEL
LIN {X 0,Y 291.957,Z 369.916,A -85,B 0,C 180,E1 -16807.349,E2 -16807.349} C_VEL
LIN {X 0,Y 293.279,Z 360.934,A -85,B 0,C 180,E1 -16809.465,E2 -16809.465} C_VEL
LIN {X 0,Y 294.581,Z 351.69,A -85,B 0,C 180,E1 -16811.213,E2 -16811.213} C_VEL
LIN {X 0,Y 295.97,Z 341.741,A -85,B 0,C 180,E1 -16812.735,E2 -16812.735} C_VEL
LIN {X 0,Y 297.276,Z 330.996,A -85,B 0,C 180,E1 -16814.05,E2 -16814.05} C_VEL
LIN {X 0,Y 298.594,Z 318.534,A -85,B 0,C 180,E1 -16815.235,E2 -16815.235} C_VEL
LIN {X 0,Y 299.482,Z 306.769,A -85,B 0,C 180,E1 -16816.083,E2 -16816.083} C_VEL
LIN {X 0,Y 300.371,Z 293.696,A -85,B 0,C 180,E1 -16816.729,E2 -16816.729} C_VEL
LIN {X 0,Y 300.993,Z 276.513,A -85,B 0,C 180,E1 -16817.229,E2 -16817.229} C_VEL
LIN {X 0,Y 302.56,Z 217.096,A -85,B 0,C 180,E1 -16818.732,E2 -16818.732} C_VEL
LIN {X 0,Y 299.264,Z 199.426,A -85,B 0,C 180,E1 -16819.463,E2 -16819.463} C_VEL
LIN {X 0,Y 293.487,Z 183.149,A -85,B 0,C 180,E1 -16820.395,E2 -16820.395} C_VEL
LIN {X 0,Y 292.74,Z 179.036,A -85,B 0,C 180,E1 -16821.72,E2 -16821.72} C_VEL
LIN {X 0,Y 291.743,Z 173.706,A -85,B 0,C 180,E1 -16823.691,E2 -16823.691} C_VEL
LIN {X 0,Y 291.887,Z 173.625,A -85,B 0,C 180,E1 -16828.622,E2 -16828.622} C_VEL
LIN {X 0,Y 291.886,Z 173.624,A -85,B 0,C 180,E1 -16831.381,E2 -16831.381} C_VEL
LIN {X 0,Y 291.721,Z 173.645,A -85,B 0,C 180,E1 -16836.92,E2 -16836.92} C_VEL
LIN {X 0,Y 291.567,Z 173.668,A -85,B 0,C 180,E1 -16839.715,E2 -16839.715} C_VEL
LIN {X 0,Y 291.521,Z 173.67,A -85,B 0,C 180,E1 -16843.952,E2 -16843.952} C_VEL
LIN {X 0,Y 291.486,Z 173.675,A -85,B 0,C 180,E1 -16846.819,E2 -16846.819} C_VEL
LIN {X 0,Y 291.45,Z 173.677,A -85,B 0,C 180,E1 -16849.876,E2 -16849.876} C_VEL
LIN {X 0,Y 291.399,Z 173.683,A -85,B 0,C 180,E1 -16854.207,E2 -16854.207} C_VEL
LIN {X 0,Y 291.418,Z 173.679,A -85,B 0,C 180,E1 -16857.273,E2 -16857.273} C_VEL
LIN {X 0,Y 291.334,Z 173.693,A -85,B 0,C 180,E1 -16860.438,E2 -16860.438} C_VEL
LIN {X 0,Y 291.345,Z 173.688,A -85,B 0,C 180,E1 -16863.7,E2 -16863.7} C_VEL
LIN {X 0,Y 291.372,Z 173.684,A -85,B 0,C 180,E1 -16867.254,E2 -16867.254} C_VEL
LIN {X 0,Y 291.333,Z 173.694,A -85,B 0,C 180,E1 -16870.644,E2 -16870.644} C_VEL
LIN {X 0,Y 291.315,Z 173.696,A -85,B 0,C 180,E1 -16874.398,E2 -16874.398} C_VEL
LIN {X 0,Y 291.326,Z 173.682,A -85,B 0,C 180,E1 -16878.406,E2 -16878.406} C_VEL
LIN {X 0,Y 291.344,Z 173.688,A -85,B 0,C 180,E1 -16881.158,E2 -16881.158} C_VEL
LIN {X 0,Y 291.356,Z 173.694,A -85,B 0,C 180,E1 -16884.626,E2 -16884.626} C_VEL
LIN {X 0,Y 291.366,Z 173.688,A -85,B 0,C 180,E1 -16887.951,E2 -16887.951} C_VEL
LIN {X 0,Y 291.345,Z 173.691,A -85,B 0,C 180,E1 -16891.155,E2 -16891.155} C_VEL
LIN {X 0,Y 291.352,Z 173.692,A -85,B 0,C 180,E1 -16892.859,E2 -16892.859} C_VEL
LIN {X 0,Y 290.674,Z 173.777,A -85,B 0,C 180,E1 -16894.013,E2 -16894.013} C_VEL
LIN {X 0,Y 287.807,Z 174.132,A -85,B 0,C 180,E1 -16895.893,E2 -16895.893} C_VEL
LIN {X 0,Y 285.398,Z 174.431,A -85,B 0,C 180,E1 -16897.42,E2 -16897.42} C_VEL
LIN {X 0,Y 284.393,Z 174.558,A -85,B 0,C 180,E1 -16898.603,E2 -16898.603} C_VEL
LIN {X 0,Y 284.325,Z 174.563,A -85,B 0,C 180,E1 -16899.003,E2 -16899.003} C_VEL
LIN {X 0,Y 284.427,Z 174.551,A -85,B 0,C 180,E1 -16902.752,E2 -16902.752} C_VEL
LIN {X 0,Y 284.48,Z 174.544,A -85,B 0,C 180,E1 -16905.698,E2 -16905.698} C_VEL
LIN {X 0,Y 284.516,Z 174.544,A -85,B 0,C 180,E1 -16910.044,E2 -16910.044} C_VEL
LIN {X 0,Y 284.644,Z 174.522,A -85,B 0,C 180,E1 -16912.909,E2 -16912.909} C_VEL
LIN {X 0,Y 284.847,Z 174.499,A -85,B 0,C 180,E1 -16918.587,E2 -16918.587} C_VEL
LIN {X 0,Y 284.841,Z 174.495,A -85,B 0,C 180,E1 -16921.414,E2 -16921.414} C_VEL
LIN {X 0,Y 284.643,Z 174.523,A -85,B 0,C 180,E1 -16927.092,E2 -16927.092} C_VEL
LIN {X 0,Y 284.517,Z 174.544,A -85,B 0,C 180,E1 -16929.958,E2 -16929.958} C_VEL
LIN {X 0,Y 284.466,Z 174.54,A -85,B 0,C 180,E1 -16934.304,E2 -16934.304} C_VEL
LIN {X 0,Y 284.332,Z 174.562,A -85,B 0,C 180,E1 -16938.744,E2 -16938.744} C_VEL
LIN {X 0,Y 284.311,Z 174.568,A -85,B 0,C 180,E1 -16943.298,E2 -16943.298} C_VEL
LIN {X 0,Y 284.329,Z 174.561,A -85,B 0,C 180,E1 -16947.145,E2 -16947.145} C_VEL
LIN {X 0,Y 284.298,Z 174.57,A -85,B 0,C 180,E1 -16950.091,E2 -16950.091} C_VEL
LIN {X 0,Y 284.308,Z 174.566,A -85,B 0,C 180,E1 -16952.946,E2 -16952.946} C_VEL
LIN {X 0,Y 284.324,Z 174.566,A -85,B 0,C 180,E1 -16956.388,E2 -16956.388} C_VEL
LIN {X 0,Y 284.286,Z 174.566,A -85,B 0,C 180,E1 -16959.999,E2 -16959.999} C_VEL
LIN {X 0,Y 284.238,Z 174.577,A -85,B 0,C 180,E1 -16964.188,E2 -16964.188} C_VEL
LIN {X 0,Y 284.243,Z 174.577,A -85,B 0,C 180,E1 -16968.118,E2 -16968.118} C_VEL
LIN {X 0,Y 284.285,Z 174.574,A -85,B 0,C 180,E1 -16972.289,E2 -16972.289} C_VEL
LIN {X 0,Y 284.311,Z 174.571,A -85,B 0,C 180,E1 -16975.35,E2 -16975.35} C_VEL
LIN {X 0,Y 284.316,Z 174.705,A -85,B 0,C 180,E1 -16977.435,E2 -16977.435} C_VEL
LIN {X 0,Y 286.446,Z 184.63,A -85,B 0,C 180,E1 -16980.962,E2 -16980.962} C_VEL
LIN {X 0,Y 287.758,Z 191.349,A -85,B 0,C 180,E1 -16983.142,E2 -16983.142} C_VEL
LIN {X 0,Y 290.879,Z 200.844,A -85,B 0,C 180,E1 -16983.718,E2 -16983.718} C_VEL
LIN {X 0,Y 295.667,Z 231.737,A -85,B 0,C 180,E1 -16984.959,E2 -16984.959} C_VEL
LIN {X 0,Y 293.763,Z 299.567,A -85,B 0,C 180,E1 -16986.749,E2 -16986.749} C_VEL
LIN {X 0,Y 292.877,Z 313.117,A -85,B 0,C 180,E1 -16987.374,E2 -16987.374} C_VEL
LIN {X 0,Y 291.745,Z 326.025,A -85,B 0,C 180,E1 -16988.26,E2 -16988.26} C_VEL
LIN {X 0,Y 290.248,Z 338.603,A -85,B 0,C 180,E1 -16989.444,E2 -16989.444} C_VEL
LIN {X 0,Y 288.788,Z 349.871,A -85,B 0,C 180,E1 -16990.819,E2 -16990.819} C_VEL
LIN {X 0,Y 287.556,Z 359.104,A -85,B 0,C 180,E1 -16992.227,E2 -16992.227} C_VEL
LIN {X 0,Y 286.291,Z 368.373,A -85,B 0,C 180,E1 -16993.967,E2 -16993.967} C_VEL
LIN {X 0,Y 284.882,Z 377.444,A -85,B 0,C 180,E1 -16996.081,E2 -16996.081} C_VEL
LIN {X 0,Y 283.818,Z 384.735,A -85,B 0,C 180,E1 -16998.211,E2 -16998.211} C_VEL
LIN {X 0,Y 283.185,Z 389.643,A -85,B 0,C 180,E1 -16999.994,E2 -16999.994} C_VEL
LIN {X 0,Y 282.689,Z 394.393,A -85,B 0,C 180,E1 -17002.14,E2 -17002.14} C_VEL
LIN {X 0,Y 282.397,Z 398.386,A -85,B 0,C 180,E1 -17004.555,E2 -17004.555} C_VEL
LIN {X 0,Y 282.302,Z 401.193,A -85,B 0,C 180,E1 -17007.145,E2 -17007.145} C_VEL
LIN {X 0,Y 282.299,Z 402.155,A -85,B 0,C 180,E1 -17008.572,E2 -17008.572} C_VEL
LIN {X 0,Y 282.306,Z 402.72,A -85,B 0,C 180,E1 -17009.999,E2 -17009.999} C_VEL
LIN {X 0,Y 282.299,Z 402.854,A -85,B 0,C 180,E1 -17011.425,E2 -17011.425} C_VEL
LIN {X 0,Y 282.307,Z 402.571,A -85,B 0,C 180,E1 -17012.852,E2 -17012.852} C_VEL
LIN {X 0,Y 282.444,Z 400.838,A -85,B 0,C 180,E1 -17015.711,E2 -17015.711} C_VEL
LIN {X 0,Y 282.66,Z 399.338,A -85,B 0,C 180,E1 -17017.14,E2 -17017.14} C_VEL
LIN {X 0,Y 283.154,Z 396.288,A -85,B 0,C 180,E1 -17019.283,E2 -17019.283} C_VEL
LIN {X 0,Y 283.922,Z 392.187,A -85,B 0,C 180,E1 -17021.42,E2 -17021.42} C_VEL
LIN {X 0,Y 285.229,Z 385.909,A -85,B 0,C 180,E1 -17023.899,E2 -17023.899} C_VEL
LIN {X 0,Y 286.906,Z 379.087,A -85,B 0,C 180,E1 -17025.995,E2 -17025.995} C_VEL
LIN {X 0,Y 288.467,Z 371.741,A -85,B 0,C 180,E1 -17027.835,E2 -17027.835} C_VEL
LIN {X 0,Y 290.08,Z 363.88,A -85,B 0,C 180,E1 -17029.457,E2 -17029.457} C_VEL
LIN {X 0,Y 292.147,Z 353.731,A -85,B 0,C 180,E1 -17031.15,E2 -17031.15} C_VEL
LIN {X 0,Y 294.29,Z 342.31,A -85,B 0,C 180,E1 -17032.647,E2 -17032.647} C_VEL
LIN {X 0,Y 296.089,Z 331.147,A -85,B 0,C 180,E1 -17033.796,E2 -17033.796} C_VEL
LIN {X 0,Y 297.726,Z 318.654,A -85,B 0,C 180,E1 -17034.769,E2 -17034.769} C_VEL
LIN {X 0,Y 299.042,Z 305.551,A -85,B 0,C 180,E1 -17035.489,E2 -17035.489} C_VEL
LIN {X 0,Y 299.766,Z 293.176,A -85,B 0,C 180,E1 -17035.936,E2 -17035.936} C_VEL
LIN {X 0,Y 301.967,Z 233.819,A -85,B 0,C 180,E1 -17037.483,E2 -17037.483} C_VEL
LIN {X 0,Y 299.085,Z 216.368,A -85,B 0,C 180,E1 -17038.388,E2 -17038.388} C_VEL
LIN {X 0,Y 297.84,Z 210.94,A -85,B 0,C 180,E1 -17038.722,E2 -17038.722} C_VEL
LIN {X 0,Y 291.966,Z 197.956,A -85,B 0,C 180,E1 -17039.937,E2 -17039.937} C_VEL
LIN {X 0,Y 288.31,Z 190.279,A -85,B 0,C 180,E1 -17040.772,E2 -17040.772} C_VEL
LIN {X 0,Y 286.403,Z 182.436,A -85,B 0,C 180,E1 -17043.782,E2 -17043.782} C_VEL
LIN {X 0,Y 284.338,Z 174.674,A -85,B 0,C 180,E1 -17047.156,E2 -17047.156} C_VEL
LIN {X 0,Y 284.25,Z 174.576,A -85,B 0,C 180,E1 -17050.001,E2 -17050.001} C_VEL
LIN {X 0,Y 284.227,Z 174.578,A -85,B 0,C 180,E1 -17054.186,E2 -17054.186} C_VEL
LIN {X 0,Y 284.232,Z 174.581,A -85,B 0,C 180,E1 -17058.116,E2 -17058.116} C_VEL
LIN {X 0,Y 284.3,Z 174.564,A -85,B 0,C 180,E1 -17062.28,E2 -17062.28} C_VEL
LIN {X 0,Y 284.299,Z 174.564,A -85,B 0,C 180,E1 -17065.349,E2 -17065.349} C_VEL
LIN {X 0,Y 284.276,Z 174.567,A -85,B 0,C 180,E1 -17068.723,E2 -17068.723} C_VEL
LIN {X 0,Y 284.273,Z 174.57,A -85,B 0,C 180,E1 -17071.982,E2 -17071.982} C_VEL
LIN {X 0,Y 284.311,Z 174.562,A -85,B 0,C 180,E1 -17076.146,E2 -17076.146} C_VEL
LIN {X 0,Y 284.324,Z 174.561,A -85,B 0,C 180,E1 -17079.927,E2 -17079.927} C_VEL
LIN {X 0,Y 284.436,Z 174.544,A -85,B 0,C 180,E1 -17084.492,E2 -17084.492} C_VEL
LIN {X 0,Y 284.455,Z 174.543,A -85,B 0,C 180,E1 -17088.6,E2 -17088.6} C_VEL
LIN {X 0,Y 284.605,Z 174.532,A -85,B 0,C 180,E1 -17091.479,E2 -17091.479} C_VEL
LIN {X 0,Y 284.565,Z 174.537,A -85,B 0,C 180,E1 -17094.33,E2 -17094.33} C_VEL
LIN {X 0,Y 284.826,Z 174.506,A -85,B 0,C 180,E1 -17098.585,E2 -17098.585} C_VEL
LIN {X 0,Y 284.834,Z 174.505,A -85,B 0,C 180,E1 -17101.413,E2 -17101.413} C_VEL
LIN {X 0,Y 284.646,Z 174.526,A -85,B 0,C 180,E1 -17107.091,E2 -17107.091} C_VEL
LIN {X 0,Y 284.501,Z 174.545,A -85,B 0,C 180,E1 -17109.957,E2 -17109.957} C_VEL
LIN {X 0,Y 284.451,Z 174.551,A -85,B 0,C 180,E1 -17114.304,E2 -17114.304} C_VEL
LIN {X 0,Y 284.321,Z 174.572,A -85,B 0,C 180,E1 -17118.743,E2 -17118.743} C_VEL
LIN {X 0,Y 284.349,Z 174.706,A -85,B 0,C 180,E1 -17119.303,E2 -17119.303} C_VEL
LIN {X 0,Y 286.692,Z 183.362,A -85,B 0,C 180,E1 -17122.997,E2 -17122.997} C_VEL
LIN {X 0,Y 289.397,Z 188.798,A -85,B 0,C 180,E1 -17123.669,E2 -17123.669} C_VEL
LIN {X 0,Y 296.181,Z 202.435,A -85,B 0,C 180,E1 -17125.064,E2 -17125.064} C_VEL
LIN {X 0,Y 301.141,Z 213.98,A -85,B 0,C 180,E1 -17126.077,E2 -17126.077} C_VEL
LIN {X 0,Y 302.468,Z 221.989,A -85,B 0,C 180,E1 -17126.493,E2 -17126.493} C_VEL
LIN {X 0,Y 299.668,Z 291.821,A -85,B 0,C 180,E1 -17128.337,E2 -17128.337} C_VEL
LIN {X 0,Y 298.61,Z 304.797,A -85,B 0,C 180,E1 -17128.932,E2 -17128.932} C_VEL
LIN {X 0,Y 297.33,Z 317.042,A -85,B 0,C 180,E1 -17129.76,E2 -17129.76} C_VEL
LIN {X 0,Y 295.687,Z 328.89,A -85,B 0,C 180,E1 -17130.841,E2 -17130.841} C_VEL
LIN {X 0,Y 293.751,Z 340.45,A -85,B 0,C 180,E1 -17132.206,E2 -17132.206} C_VEL
LIN {X 0,Y 291.936,Z 349.993,A -85,B 0,C 180,E1 -17133.62,E2 -17133.62} C_VEL
LIN {X 0,Y 290.032,Z 358.801,A -85,B 0,C 180,E1 -17135.216,E2 -17135.216} C_VEL
LIN {X 0,Y 288.16,Z 367.354,A -85,B 0,C 180,E1 -17137.149,E2 -17137.149} C_VEL
LIN {X 0,Y 286.521,Z 374.351,A -85,B 0,C 180,E1 -17139.105,E2 -17139.105} C_VEL
LIN {X 0,Y 285.199,Z 380.113,A -85,B 0,C 180,E1 -17141.101,E2 -17141.101} C_VEL
LIN {X 0,Y 284.171,Z 384.723,A -85,B 0,C 180,E1 -17143.102,E2 -17143.102} C_VEL
LIN {X 0,Y 283.407,Z 388.224,A -85,B 0,C 180,E1 -17145.032,E2 -17145.032} C_VEL
LIN {X 0,Y 282.862,Z 390.838,A -85,B 0,C 180,E1 -17146.946,E2 -17146.946} C_VEL
LIN {X 0,Y 282.283,Z 393.219,A -85,B 0,C 180,E1 -17149.663,E2 -17149.663} C_VEL
LIN {X 0,Y 282.037,Z 393.998,A -85,B 0,C 180,E1 -17151.469,E2 -17151.469} C_VEL
LIN {X 0,Y 281.979,Z 394.11,A -85,B 0,C 180,E1 -17153.263,E2 -17153.263} C_VEL
LIN {X 0,Y 281.949,Z 393.471,A -85,B 0,C 180,E1 -17155.342,E2 -17155.342} C_VEL
LIN {X 0,Y 282.143,Z 391.499,A -85,B 0,C 180,E1 -17157.877,E2 -17157.877} C_VEL
LIN {X 0,Y 282.603,Z 388.051,A -85,B 0,C 180,E1 -17160.505,E2 -17160.505} C_VEL
LIN {X 0,Y 283.082,Z 384.111,A -85,B 0,C 180,E1 -17162.619,E2 -17162.619} C_VEL
LIN {X 0,Y 283.739,Z 379.091,A -85,B 0,C 180,E1 -17164.708,E2 -17164.708} C_VEL
LIN {X 0,Y 284.757,Z 371.617,A -85,B 0,C 180,E1 -17167.127,E2 -17167.127} C_VEL
LIN {X 0,Y 285.856,Z 363.911,A -85,B 0,C 180,E1 -17169.107,E2 -17169.107} C_VEL
LIN {X 0,Y 287.347,Z 354.284,A -85,B 0,C 180,E1 -17171.093,E2 -17171.093} C_VEL
LIN {X 0,Y 288.742,Z 344.398,A -85,B 0,C 180,E1 -17172.718,E2 -17172.718} C_VEL
LIN {X 0,Y 290.23,Z 333.188,A -85,B 0,C 180,E1 -17174.193,E2 -17174.193} C_VEL
LIN {X 0,Y 291.549,Z 321.419,A -85,B 0,C 180,E1 -17175.405,E2 -17175.405} C_VEL
LIN {X 0,Y 292.595,Z 309.006,A -85,B 0,C 180,E1 -17176.369,E2 -17176.369} C_VEL
LIN {X 0,Y 293.568,Z 296.046,A -85,B 0,C 180,E1 -17177.076,E2 -17177.076} C_VEL
LIN {X 0,Y 294.109,Z 282.305,A -85,B 0,C 180,E1 -17177.539,E2 -17177.539} C_VEL
LIN {X 0,Y 295.875,Z 217.573,A -85,B 0,C 180,E1 -17179.214,E2 -17179.214} C_VEL
LIN {X 0,Y 292.943,Z 201.879,A -85,B 0,C 180,E1 -17179.882,E2 -17179.882} C_VEL
LIN {X 0,Y 286.304,Z 183.142,A -85,B 0,C 180,E1 -17180.998,E2 -17180.998} C_VEL
LIN {X 0,Y 284.914,Z 175.611,A -85,B 0,C 180,E1 -17183.629,E2 -17183.629} C_VEL
LIN {X 0,Y 284.627,Z 174.556,A -85,B 0,C 180,E1 -17184.156,E2 -17184.156} C_VEL
LIN {X 0,Y 284.853,Z 174.501,A -85,B 0,C 180,E1 -17188.588,E2 -17188.588} C_VEL
LIN {X 0,Y 284.852,Z 174.5,A -85,B 0,C 180,E1 -17191.415,E2 -17191.415} C_VEL
LIN {X 0,Y 284.672,Z 174.524,A -85,B 0,C 180,E1 -17197.092,E2 -17197.092} C_VEL
LIN {X 0,Y 284.512,Z 174.545,A -85,B 0,C 180,E1 -17199.959,E2 -17199.959} C_VEL
LIN {X 0,Y 284.481,Z 174.546,A -85,B 0,C 180,E1 -17204.304,E2 -17204.304} C_VEL
LIN {X 0,Y 284.425,Z 174.555,A -85,B 0,C 180,E1 -17207.25,E2 -17207.25} C_VEL
LIN {X 0,Y 284.378,Z 174.557,A -85,B 0,C 180,E1 -17210.243,E2 -17210.243} C_VEL
LIN {X 0,Y 284.369,Z 174.559,A -85,B 0,C 180,E1 -17213.876,E2 -17213.876} C_VEL
LIN {X 0,Y 284.394,Z 174.552,A -85,B 0,C 180,E1 -17217.174,E2 -17217.174} C_VEL
LIN {X 0,Y 284.294,Z 174.573,A -85,B 0,C 180,E1 -17221.276,E2 -17221.276} C_VEL
LIN {X 0,Y 284.341,Z 174.554,A -85,B 0,C 180,E1 -17225.349,E2 -17225.349} C_VEL
LIN {X 0,Y 284.308,Z 174.561,A -85,B 0,C 180,E1 -17228.171,E2 -17228.171} C_VEL
LIN {X 0,Y 284.27,Z 174.573,A -85,B 0,C 180,E1 -17232.126,E2 -17232.126} C_VEL
LIN {X 0,Y 284.27,Z 174.568,A -85,B 0,C 180,E1 -17236.193,E2 -17236.193} C_VEL
LIN {X 0,Y 284.307,Z 174.556,A -85,B 0,C 180,E1 -17240.025,E2 -17240.025} C_VEL
LIN {X 0,Y 284.322,Z 174.565,A -85,B 0,C 180,E1 -17243.613,E2 -17243.613} C_VEL
LIN {X 0,Y 284.307,Z 174.567,A -85,B 0,C 180,E1 -17247.191,E2 -17247.191} C_VEL
LIN {X 0,Y 284.338,Z 174.565,A -85,B 0,C 180,E1 -17250.374,E2 -17250.374} C_VEL
LIN {X 0,Y 284.308,Z 174.568,A -85,B 0,C 180,E1 -17253.58,E2 -17253.58} C_VEL
LIN {X 0,Y 284.332,Z 174.562,A -85,B 0,C 180,E1 -17256.705,E2 -17256.705} C_VEL
LIN {X 0,Y 284.325,Z 174.563,A -85,B 0,C 180,E1 -17259.003,E2 -17259.003} C_VEL
LIN {X 0,Y 283.702,Z 174.647,A -85,B 0,C 180,E1 -17260.185,E2 -17260.185} C_VEL
LIN {X 0,Y 280.891,Z 174.997,A -85,B 0,C 180,E1 -17262.112,E2 -17262.112} C_VEL
LIN {X 0,Y 278.501,Z 175.29,A -85,B 0,C 180,E1 -17263.677,E2 -17263.677} C_VEL
LIN {X 0,Y 277.498,Z 175.412,A -85,B 0,C 180,E1 -17264.889,E2 -17264.889} C_VEL
LIN {X 0,Y 277.43,Z 175.42,A -85,B 0,C 180,E1 -17265.3,E2 -17265.3} C_VEL
LIN {X 0,Y 277.46,Z 175.423,A -85,B 0,C 180,E1 -17269.788,E2 -17269.788} C_VEL
LIN {X 0,Y 277.602,Z 175.399,A -85,B 0,C 180,E1 -17272.728,E2 -17272.728} C_VEL
LIN {X 0,Y 277.813,Z 175.375,A -85,B 0,C 180,E1 -17278.551,E2 -17278.551} C_VEL
LIN {X 0,Y 277.808,Z 175.369,A -85,B 0,C 180,E1 -17281.45,E2 -17281.45} C_VEL
LIN {X 0,Y 277.602,Z 175.4,A -85,B 0,C 180,E1 -17287.273,E2 -17287.273} C_VEL
LIN {X 0,Y 277.461,Z 175.422,A -85,B 0,C 180,E1 -17290.214,E2 -17290.214} C_VEL
LIN {X 0,Y 277.412,Z 175.418,A -85,B 0,C 180,E1 -17294.676,E2 -17294.676} C_VEL
LIN {X 0,Y 277.286,Z 175.442,A -85,B 0,C 180,E1 -17299.239,E2 -17299.239} C_VEL
LIN {X 0,Y 277.258,Z 175.442,A -85,B 0,C 180,E1 -17303.928,E2 -17303.928} C_VEL
LIN {X 0,Y 277.27,Z 175.443,A -85,B 0,C 180,E1 -17307.481,E2 -17307.481} C_VEL
LIN {X 0,Y 277.252,Z 175.448,A -85,B 0,C 180,E1 -17310.473,E2 -17310.473} C_VEL
LIN {X 0,Y 277.25,Z 175.44,A -85,B 0,C 180,E1 -17313.896,E2 -17313.896} C_VEL
LIN {X 0,Y 277.258,Z 175.447,A -85,B 0,C 180,E1 -17317.472,E2 -17317.472} C_VEL
LIN {X 0,Y 277.188,Z 175.457,A -85,B 0,C 180,E1 -17321.241,E2 -17321.241} C_VEL
LIN {X 0,Y 277.178,Z 175.455,A -85,B 0,C 180,E1 -17325.232,E2 -17325.232} C_VEL
LIN {X 0,Y 277.181,Z 175.458,A -85,B 0,C 180,E1 -17328.757,E2 -17328.757} C_VEL
LIN {X 0,Y 277.236,Z 175.453,A -85,B 0,C 180,E1 -17332.524,E2 -17332.524} C_VEL
LIN {X 0,Y 277.25,Z 175.451,A -85,B 0,C 180,E1 -17336.103,E2 -17336.103} C_VEL
LIN {X 0,Y 277.285,Z 175.584,A -85,B 0,C 180,E1 -17337.012,E2 -17337.012} C_VEL
LIN {X 0,Y 279.418,Z 185.51,A -85,B 0,C 180,E1 -17340.627,E2 -17340.627} C_VEL
LIN {X 0,Y 280.504,Z 191.23,A -85,B 0,C 180,E1 -17342.533,E2 -17342.533} C_VEL
LIN {X 0,Y 284.408,Z 202.448,A -85,B 0,C 180,E1 -17343.244,E2 -17343.244} C_VEL
LIN {X 0,Y 289.03,Z 232.927,A -85,B 0,C 180,E1 -17344.499,E2 -17344.499} C_VEL
LIN {X 0,Y 287.035,Z 299.976,A -85,B 0,C 180,E1 -17346.314,E2 -17346.314} C_VEL
LIN {X 0,Y 286.113,Z 313.351,A -85,B 0,C 180,E1 -17346.952,E2 -17346.952} C_VEL
LIN {X 0,Y 285.026,Z 325.64,A -85,B 0,C 180,E1 -17347.816,E2 -17347.816} C_VEL
LIN {X 0,Y 283.584,Z 337.486,A -85,B 0,C 180,E1 -17348.938,E2 -17348.938} C_VEL
LIN {X 0,Y 282.099,Z 348.941,A -85,B 0,C 180,E1 -17350.345,E2 -17350.345} C_VEL
LIN {X 0,Y 280.621,Z 359.284,A -85,B 0,C 180,E1 -17351.945,E2 -17351.945} C_VEL
LIN {X 0,Y 279.151,Z 369.391,A -85,B 0,C 180,E1 -17353.921,E2 -17353.921} C_VEL
LIN {X 0,Y 277.749,Z 378.275,A -85,B 0,C 180,E1 -17356.09,E2 -17356.09} C_VEL
LIN {X 0,Y 276.68,Z 385.341,A -85,B 0,C 180,E1 -17358.274,E2 -17358.274} C_VEL
LIN {X 0,Y 275.957,Z 390.984,A -85,B 0,C 180,E1 -17360.47,E2 -17360.47} C_VEL
LIN {X 0,Y 275.511,Z 395.396,A -85,B 0,C 180,E1 -17362.671,E2 -17362.671} C_VEL
LIN {X 0,Y 275.311,Z 398.382,A -85,B 0,C 180,E1 -17364.613,E2 -17364.613} C_VEL
LIN {X 0,Y 275.215,Z 400.996,A -85,B 0,C 180,E1 -17367.071,E2 -17367.071} C_VEL
LIN {X 0,Y 275.225,Z 401.983,A -85,B 0,C 180,E1 -17368.535,E2 -17368.535} C_VEL
LIN {X 0,Y 275.23,Z 402.573,A -85,B 0,C 180,E1 -17369.998,E2 -17369.998} C_VEL
LIN {X 0,Y 275.225,Z 402.753,A -85,B 0,C 180,E1 -17371.462,E2 -17371.462} C_VEL
LIN {X 0,Y 275.22,Z 402.495,A -85,B 0,C 180,E1 -17372.926,E2 -17372.926} C_VEL
LIN {X 0,Y 275.382,Z 400.808,A -85,B 0,C 180,E1 -17375.858,E2 -17375.858} C_VEL
LIN {X 0,Y 275.603,Z 399.355,A -85,B 0,C 180,E1 -17377.324,E2 -17377.324} C_VEL
LIN {X 0,Y 276.137,Z 396.348,A -85,B 0,C 180,E1 -17379.521,E2 -17379.521} C_VEL
LIN {X 0,Y 276.958,Z 392.301,A -85,B 0,C 180,E1 -17381.711,E2 -17381.711} C_VEL
LIN {X 0,Y 278.328,Z 386.109,A -85,B 0,C 180,E1 -17384.251,E2 -17384.251} C_VEL
LIN {X 0,Y 280.101,Z 379.373,A -85,B 0,C 180,E1 -17386.394,E2 -17386.394} C_VEL
LIN {X 0,Y 281.497,Z 373.311,A -85,B 0,C 180,E1 -17387.988,E2 -17387.988} C_VEL
LIN {X 0,Y 283.04,Z 366.121,A -85,B 0,C 180,E1 -17389.583,E2 -17389.583} C_VEL
LIN {X 0,Y 285.136,Z 356.492,A -85,B 0,C 180,E1 -17391.317,E2 -17391.317} C_VEL
LIN {X 0,Y 287.23,Z 345.852,A -85,B 0,C 180,E1 -17392.855,E2 -17392.855} C_VEL
LIN {X 0,Y 289.138,Z 335.587,A -85,B 0,C 180,E1 -17394.023,E2 -17394.023} C_VEL
LIN {X 0,Y 290.949,Z 323.412,A -85,B 0,C 180,E1 -17395.1,E2 -17395.1} C_VEL
LIN {X 0,Y 292.497,Z 310.106,A -85,B 0,C 180,E1 -17395.959,E2 -17395.959} C_VEL
LIN {X 0,Y 293.5,Z 296.729,A -85,B 0,C 180,E1 -17396.532,E2 -17396.532} C_VEL
LIN {X 0,Y 296.028,Z 235.32,A -85,B 0,C 180,E1 -17398.176,E2 -17398.176} C_VEL
LIN {X 0,Y 293.484,Z 219.237,A -85,B 0,C 180,E1 -17399.029,E2 -17399.029} C_VEL
LIN {X 0,Y 292.268,Z 213.886,A -85,B 0,C 180,E1 -17399.368,E2 -17399.368} C_VEL
LIN {X 0,Y 286.386,Z 200.873,A -85,B 0,C 180,E1 -17400.643,E2 -17400.643} C_VEL
LIN {X 0,Y 282.59,Z 193.359,A -85,B 0,C 180,E1 -17401.498,E2 -17401.498} C_VEL
LIN {X 0,Y 281.043,Z 189.945,A -85,B 0,C 180,E1 -17401.934,E2 -17401.934} C_VEL
LIN {X 0,Y 278.893,Z 181.47,A -85,B 0,C 180,E1 -17405.419,E2 -17405.419} C_VEL
LIN {X 0,Y 277.24,Z 175.488,A -85,B 0,C 180,E1 -17408.245,E2 -17408.245} C_VEL
LIN {X 0,Y 277.186,Z 175.458,A -85,B 0,C 180,E1 -17412.667,E2 -17412.667} C_VEL
LIN {X 0,Y 277.184,Z 175.455,A -85,B 0,C 180,E1 -17416.796,E2 -17416.796} C_VEL
LIN {X 0,Y 277.209,Z 175.455,A -85,B 0,C 180,E1 -17420.667,E2 -17420.667} C_VEL
LIN {X 0,Y 277.27,Z 175.448,A -85,B 0,C 180,E1 -17424.339,E2 -17424.339} C_VEL
LIN {X 0,Y 277.231,Z 175.45,A -85,B 0,C 180,E1 -17427.834,E2 -17427.834} C_VEL
LIN {X 0,Y 277.23,Z 175.452,A -85,B 0,C 180,E1 -17431.205,E2 -17431.205} C_VEL
LIN {X 0,Y 277.236,Z 175.451,A -85,B 0,C 180,E1 -17434.471,E2 -17434.471} C_VEL
LIN {X 0,Y 277.249,Z 175.443,A -85,B 0,C 180,E1 -17437.651,E2 -17437.651} C_VEL
LIN {X 0,Y 277.275,Z 175.435,A -85,B 0,C 180,E1 -17440.76,E2 -17440.76} C_VEL
LIN {X 0,Y 277.399,Z 175.421,A -85,B 0,C 180,E1 -17445.323,E2 -17445.323} C_VEL
LIN {X 0,Y 277.444,Z 175.42,A -85,B 0,C 180,E1 -17449.786,E2 -17449.786} C_VEL
LIN {X 0,Y 277.599,Z 175.397,A -85,B 0,C 180,E1 -17452.727,E2 -17452.727} C_VEL
LIN {X 0,Y 277.793,Z 175.382,A -85,B 0,C 180,E1 -17458.55,E2 -17458.55} C_VEL
LIN {X 0,Y 277.8,Z 175.381,A -85,B 0,C 180,E1 -17461.449,E2 -17461.449} C_VEL
LIN {X 0,Y 277.603,Z 175.405,A -85,B 0,C 180,E1 -17467.272,E2 -17467.272} C_VEL
LIN {X 0,Y 277.442,Z 175.426,A -85,B 0,C 180,E1 -17470.213,E2 -17470.213} C_VEL
LIN {X 0,Y 277.397,Z 175.431,A -85,B 0,C 180,E1 -17474.675,E2 -17474.675} C_VEL
LIN {X 0,Y 277.306,Z 175.565,A -85,B 0,C 180,E1 -17478.277,E2 -17478.277} C_VEL
LIN {X 0,Y 279.369,Z 183.315,A -85,B 0,C 180,E1 -17481.78,E2 -17481.78} C_VEL
LIN {X 0,Y 279.902,Z 184.651,A -85,B 0,C 180,E1 -17482.027,E2 -17482.027} C_VEL
LIN {X 0,Y 284.828,Z 193.607,A -85,B 0,C 180,E1 -17483.147,E2 -17483.147} C_VEL
LIN {X 0,Y 292.002,Z 208.446,A -85,B 0,C 180,E1 -17484.696,E2 -17484.696} C_VEL
LIN {X 0,Y 295.591,Z 217.114,A -85,B 0,C 180,E1 -17485.46,E2 -17485.46} C_VEL
LIN {X 0,Y 296.528,Z 222.74,A -85,B 0,C 180,E1 -17485.763,E2 -17485.763} C_VEL
LIN {X 0,Y 293.589,Z 291.737,A -85,B 0,C 180,E1 -17487.627,E2 -17487.627} C_VEL
LIN {X 0,Y 292.487,Z 304.836,A -85,B 0,C 180,E1 -17488.238,E2 -17488.238} C_VEL
LIN {X 0,Y 291.048,Z 317.784,A -85,B 0,C 180,E1 -17489.137,E2 -17489.137} C_VEL
LIN {X 0,Y 289.413,Z 328.867,A -85,B 0,C 180,E1 -17490.169,E2 -17490.169} C_VEL
LIN {X 0,Y 287.512,Z 339.827,A -85,B 0,C 180,E1 -17491.475,E2 -17491.475} C_VEL
LIN {X 0,Y 285.341,Z 350.83,A -85,B 0,C 180,E1 -17493.135,E2 -17493.135} C_VEL
LIN {X 0,Y 283.088,Z 360.563,A -85,B 0,C 180,E1 -17494.993,E2 -17494.993} C_VEL
LIN {X 0,Y 281.234,Z 368.57,A -85,B 0,C 180,E1 -17496.905,E2 -17496.905} C_VEL
LIN {X 0,Y 279.538,Z 375.476,A -85,B 0,C 180,E1 -17498.941,E2 -17498.941} C_VEL
LIN {X 0,Y 278.094,Z 381.263,A -85,B 0,C 180,E1 -17501.076,E2 -17501.076} C_VEL
LIN {X 0,Y 277.005,Z 385.856,A -85,B 0,C 180,E1 -17503.237,E2 -17503.237} C_VEL
LIN {X 0,Y 276.176,Z 389.42,A -85,B 0,C 180,E1 -17505.44,E2 -17505.44} C_VEL
LIN {X 0,Y 275.56,Z 392.017,A -85,B 0,C 180,E1 -17507.699,E2 -17507.699} C_VEL
LIN {X 0,Y 275.099,Z 393.792,A -85,B 0,C 180,E1 -17510.309,E2 -17510.309} C_VEL
LIN {X 0,Y 274.881,Z 394.261,A -85,B 0,C 180,E1 -17512.427,E2 -17512.427} C_VEL
LIN {X 0,Y 274.843,Z 393.764,A -85,B 0,C 180,E1 -17514.911,E2 -17514.911} C_VEL
LIN {X 0,Y 275.002,Z 391.936,A -85,B 0,C 180,E1 -17517.545,E2 -17517.545} C_VEL
LIN {X 0,Y 275.458,Z 388.748,A -85,B 0,C 180,E1 -17520.165,E2 -17520.165} C_VEL
LIN {X 0,Y 276.02,Z 384.227,A -85,B 0,C 180,E1 -17522.724,E2 -17522.724} C_VEL
LIN {X 0,Y 276.76,Z 378.233,A -85,B 0,C 180,E1 -17525.227,E2 -17525.227} C_VEL
LIN {X 0,Y 277.729,Z 371.882,A -85,B 0,C 180,E1 -17527.302,E2 -17527.302} C_VEL
LIN {X 0,Y 278.855,Z 364.168,A -85,B 0,C 180,E1 -17529.341,E2 -17529.341} C_VEL
LIN {X 0,Y 280.309,Z 355.256,A -85,B 0,C 180,E1 -17531.242,E2 -17531.242} C_VEL
LIN {X 0,Y 281.759,Z 345.262,A -85,B 0,C 180,E1 -17532.959,E2 -17532.959} C_VEL
LIN {X 0,Y 283.196,Z 334.929,A -85,B 0,C 180,E1 -17534.381,E2 -17534.381} C_VEL
LIN {X 0,Y 284.62,Z 322.753,A -85,B 0,C 180,E1 -17535.706,E2 -17535.706} C_VEL
LIN {X 0,Y 285.702,Z 311.127,A -85,B 0,C 180,E1 -17536.668,E2 -17536.668} C_VEL
LIN {X 0,Y 286.718,Z 297.941,A -85,B 0,C 180,E1 -17537.442,E2 -17537.442} C_VEL
LIN {X 0,Y 287.357,Z 285.293,A -85,B 0,C 180,E1 -17537.919,E2 -17537.919} C_VEL
LIN {X 0,Y 289.255,Z 218.53,A -85,B 0,C 180,E1 -17539.692,E2 -17539.692} C_VEL
LIN {X 0,Y 286.517,Z 203.939,A -85,B 0,C 180,E1 -17540.336,E2 -17540.336} C_VEL
LIN {X 0,Y 279.234,Z 183.507,A -85,B 0,C 180,E1 -17541.589,E2 -17541.589} C_VEL
LIN {X 0,Y 278.869,Z 181.872,A -85,B 0,C 180,E1 -17542.034,E2 -17542.034} C_VEL
LIN {X 0,Y 277.576,Z 175.481,A -85,B 0,C 180,E1 -17544.508,E2 -17544.508} C_VEL
LIN {X 0,Y 277.819,Z 175.378,A -85,B 0,C 180,E1 -17548.552,E2 -17548.552} C_VEL
LIN {X 0,Y 277.818,Z 175.376,A -85,B 0,C 180,E1 -17551.451,E2 -17551.451} C_VEL
LIN {X 0,Y 277.626,Z 175.402,A -85,B 0,C 180,E1 -17557.273,E2 -17557.273} C_VEL
LIN {X 0,Y 277.456,Z 175.423,A -85,B 0,C 180,E1 -17560.215,E2 -17560.215} C_VEL
LIN {X 0,Y 277.434,Z 175.424,A -85,B 0,C 180,E1 -17564.675,E2 -17564.675} C_VEL
LIN {X 0,Y 277.344,Z 175.431,A -85,B 0,C 180,E1 -17569.235,E2 -17569.235} C_VEL
LIN {X 0,Y 277.318,Z 175.437,A -85,B 0,C 180,E1 -17574.171,E2 -17574.171} C_VEL
LIN {X 0,Y 277.323,Z 175.435,A -85,B 0,C 180,E1 -17577.505,E2 -17577.505} C_VEL
LIN {X 0,Y 277.272,Z 175.445,A -85,B 0,C 180,E1 -17580.483,E2 -17580.483} C_VEL
LIN {X 0,Y 277.247,Z 175.443,A -85,B 0,C 180,E1 -17583.897,E2 -17583.897} C_VEL
LIN {X 0,Y 277.265,Z 175.439,A -85,B 0,C 180,E1 -17587.471,E2 -17587.471} C_VEL
LIN {X 0,Y 277.21,Z 175.454,A -85,B 0,C 180,E1 -17591.238,E2 -17591.238} C_VEL
LIN {X 0,Y 277.218,Z 175.446,A -85,B 0,C 180,E1 -17595.224,E2 -17595.224} C_VEL
LIN {X 0,Y 277.223,Z 175.437,A -85,B 0,C 180,E1 -17599.513,E2 -17599.513} C_VEL
LIN {X 0,Y 277.257,Z 175.445,A -85,B 0,C 180,E1 -17602.53,E2 -17602.53} C_VEL
LIN {X 0,Y 277.247,Z 175.449,A -85,B 0,C 180,E1 -17606.105,E2 -17606.105} C_VEL
LIN {X 0,Y 277.263,Z 175.441,A -85,B 0,C 180,E1 -17609.54,E2 -17609.54} C_VEL
LIN {X 0,Y 277.294,Z 175.443,A -85,B 0,C 180,E1 -17612.858,E2 -17612.858} C_VEL
LIN {X 0,Y 277.287,Z 175.443,A -85,B 0,C 180,E1 -17616.076,E2 -17616.076} C_VEL
LIN {X 0,Y 277.347,Z 175.435,A -85,B 0,C 180,E1 -17620.767,E2 -17620.767} C_VEL
LIN {X 0,Y 277.43,Z 175.42,A -85,B 0,C 180,E1 -17625.3,E2 -17625.3} C_VEL
LIN {X 0,Y 276.805,Z 175.503,A -85,B 0,C 180,E1 -17626.512,E2 -17626.512} C_VEL
LIN {X 0,Y 273.998,Z 175.853,A -85,B 0,C 180,E1 -17628.488,E2 -17628.488} C_VEL
LIN {X 0,Y 271.607,Z 176.151,A -85,B 0,C 180,E1 -17630.094,E2 -17630.094} C_VEL
LIN {X 0,Y 270.597,Z 176.273,A -85,B 0,C 180,E1 -17631.338,E2 -17631.338} C_VEL
LIN {X 0,Y 270.524,Z 176.279,A -85,B 0,C 180,E1 -17631.759,E2 -17631.759} C_VEL
LIN {X 0,Y 270.511,Z 176.288,A -85,B 0,C 180,E1 -17634.036,E2 -17634.036} C_VEL
LIN {X 0,Y 270.778,Z 176.251,A -85,B 0,C 180,E1 -17638.513,E2 -17638.513} C_VEL
LIN {X 0,Y 270.773,Z 176.243,A -85,B 0,C 180,E1 -17641.488,E2 -17641.488} C_VEL
LIN {X 0,Y 270.564,Z 176.278,A -85,B 0,C 180,E1 -17647.463,E2 -17647.463} C_VEL
LIN {X 0,Y 270.413,Z 176.299,A -85,B 0,C 180,E1 -17650.483,E2 -17650.483} C_VEL
LIN {X 0,Y 270.372,Z 176.293,A -85,B 0,C 180,E1 -17655.067,E2 -17655.067} C_VEL
LIN {X 0,Y 270.226,Z 176.324,A -85,B 0,C 180,E1 -17659.762,E2 -17659.762} C_VEL
LIN {X 0,Y 270.186,Z 176.322,A -85,B 0,C 180,E1 -17664.436,E2 -17664.436} C_VEL
LIN {X 0,Y 270.199,Z 176.323,A -85,B 0,C 180,E1 -17667.917,E2 -17667.917} C_VEL
LIN {X 0,Y 270.177,Z 176.329,A -85,B 0,C 180,E1 -17671.35,E2 -17671.35} C_VEL
LIN {X 0,Y 270.202,Z 176.321,A -85,B 0,C 180,E1 -17674.906,E2 -17674.906} C_VEL
LIN {X 0,Y 270.203,Z 176.326,A -85,B 0,C 180,E1 -17678.71,E2 -17678.71} C_VEL
LIN {X 0,Y 270.152,Z 176.333,A -85,B 0,C 180,E1 -17683.245,E2 -17683.245} C_VEL
LIN {X 0,Y 270.155,Z 176.332,A -85,B 0,C 180,E1 -17687.437,E2 -17687.437} C_VEL
LIN {X 0,Y 270.156,Z 176.333,A -85,B 0,C 180,E1 -17691.364,E2 -17691.364} C_VEL
LIN {X 0,Y 270.201,Z 176.327,A -85,B 0,C 180,E1 -17695.093,E2 -17695.093} C_VEL
LIN {X 0,Y 270.254,Z 176.548,A -85,B 0,C 180,E1 -17696.619,E2 -17696.619} C_VEL
LIN {X 0,Y 272.579,Z 187.461,A -85,B 0,C 180,E1 -17700.666,E2 -17700.666} C_VEL
LIN {X 0,Y 273.316,Z 191.222,A -85,B 0,C 180,E1 -17701.912,E2 -17701.912} C_VEL
LIN {X 0,Y 278.078,Z 205.056,A -85,B 0,C 180,E1 -17702.788,E2 -17702.788} C_VEL
LIN {X 0,Y 282.406,Z 233.581,A -85,B 0,C 180,E1 -17704.001,E2 -17704.001} C_VEL
LIN {X 0,Y 280.392,Z 299.29,A -85,B 0,C 180,E1 -17705.816,E2 -17705.816} C_VEL
LIN {X 0,Y 279.443,Z 312.84,A -85,B 0,C 180,E1 -17706.467,E2 -17706.467} C_VEL
LIN {X 0,Y 278.301,Z 325.239,A -85,B 0,C 180,E1 -17707.348,E2 -17707.348} C_VEL
LIN {X 0,Y 276.945,Z 336.369,A -85,B 0,C 180,E1 -17708.409,E2 -17708.409} C_VEL
LIN {X 0,Y 275.38,Z 348.003,A -85,B 0,C 180,E1 -17709.845,E2 -17709.845} C_VEL
LIN {X 0,Y 273.806,Z 358.499,A -85,B 0,C 180,E1 -17711.479,E2 -17711.479} C_VEL
LIN {X 0,Y 272.589,Z 367.178,A -85,B 0,C 180,E1 -17713.156,E2 -17713.156} C_VEL
LIN {X 0,Y 271.321,Z 374.987,A -85,B 0,C 180,E1 -17714.986,E2 -17714.986} C_VEL
LIN {X 0,Y 270.002,Z 382.673,A -85,B 0,C 180,E1 -17717.216,E2 -17717.216} C_VEL
LIN {X 0,Y 269.153,Z 388.851,A -85,B 0,C 180,E1 -17719.467,E2 -17719.467} C_VEL
LIN {X 0,Y 268.565,Z 393.726,A -85,B 0,C 180,E1 -17721.723,E2 -17721.723} C_VEL
LIN {X 0,Y 268.232,Z 397.444,A -85,B 0,C 180,E1 -17723.983,E2 -17723.983} C_VEL
LIN {X 0,Y 268.145,Z 399.358,A -85,B 0,C 180,E1 -17725.489,E2 -17725.489} C_VEL
LIN {X 0,Y 268.129,Z 400.799,A -85,B 0,C 180,E1 -17726.994,E2 -17726.994} C_VEL
LIN {X 0,Y 268.13,Z 401.811,A -85,B 0,C 180,E1 -17728.496,E2 -17728.496} C_VEL
LIN {X 0,Y 268.156,Z 402.425,A -85,B 0,C 180,E1 -17729.998,E2 -17729.998} C_VEL
LIN {X 0,Y 268.131,Z 402.642,A -85,B 0,C 180,E1 -17731.5,E2 -17731.5} C_VEL
LIN {X 0,Y 268.117,Z 402.419,A -85,B 0,C 180,E1 -17733.003,E2 -17733.003} C_VEL
LIN {X 0,Y 268.306,Z 400.782,A -85,B 0,C 180,E1 -17736.013,E2 -17736.013} C_VEL
LIN {X 0,Y 268.542,Z 399.372,A -85,B 0,C 180,E1 -17737.517,E2 -17737.517} C_VEL
LIN {X 0,Y 269.135,Z 396.415,A -85,B 0,C 180,E1 -17739.771,E2 -17739.771} C_VEL
LIN {X 0,Y 270.007,Z 392.43,A -85,B 0,C 180,E1 -17742.017,E2 -17742.017} C_VEL
LIN {X 0,Y 271.451,Z 386.33,A -85,B 0,C 180,E1 -17744.62,E2 -17744.62} C_VEL
LIN {X 0,Y 273.316,Z 379.663,A -85,B 0,C 180,E1 -17746.813,E2 -17746.813} C_VEL
LIN {X 0,Y 274.941,Z 372.396,A -85,B 0,C 180,E1 -17748.767,E2 -17748.767} C_VEL
LIN {X 0,Y 277.22,Z 363.016,A -85,B 0,C 180,E1 -17750.787,E2 -17750.787} C_VEL
LIN {X 0,Y 279.574,Z 352.693,A -85,B 0,C 180,E1 -17752.54,E2 -17752.54} C_VEL
LIN {X 0,Y 281.619,Z 342.551,A -85,B 0,C 180,E1 -17753.922,E2 -17753.922} C_VEL
LIN {X 0,Y 283.552,Z 331.541,A -85,B 0,C 180,E1 -17755.114,E2 -17755.114} C_VEL
LIN {X 0,Y 285.328,Z 319.38,A -85,B 0,C 180,E1 -17756.12,E2 -17756.12} C_VEL
LIN {X 0,Y 286.854,Z 305.841,A -85,B 0,C 180,E1 -17756.901,E2 -17756.901} C_VEL
LIN {X 0,Y 287.716,Z 292.514,A -85,B 0,C 180,E1 -17757.404,E2 -17757.404} C_VEL
LIN {X 0,Y 290.073,Z 236.017,A -85,B 0,C 180,E1 -17758.936,E2 -17758.936} C_VEL
LIN {X 0,Y 287.409,Z 219.607,A -85,B 0,C 180,E1 -17759.851,E2 -17759.851} C_VEL
LIN {X 0,Y 286.559,Z 216.428,A -85,B 0,C 180,E1 -17760.083,E2 -17760.083} C_VEL
LIN {X 0,Y 280.073,Z 202.043,A -85,B 0,C 180,E1 -17761.58,E2 -17761.58} C_VEL
LIN {X 0,Y 274.955,Z 192.369,A -85,B 0,C 180,E1 -17762.788,E2 -17762.788} C_VEL
LIN {X 0,Y 273.764,Z 189.739,A -85,B 0,C 180,E1 -17763.179,E2 -17763.179} C_VEL
LIN {X 0,Y 271.827,Z 182.101,A -85,B 0,C 180,E1 -17766.486,E2 -17766.486} C_VEL
LIN {X 0,Y 270.167,Z 176.39,A -85,B 0,C 180,E1 -17769.348,E2 -17769.348} C_VEL
LIN {X 0,Y 270.142,Z 176.338,A -85,B 0,C 180,E1 -17773.243,E2 -17773.243} C_VEL
LIN {X 0,Y 270.144,Z 176.334,A -85,B 0,C 180,E1 -17777.436,E2 -17777.436} C_VEL
LIN {X 0,Y 270.201,Z 176.326,A -85,B 0,C 180,E1 -17781.372,E2 -17781.372} C_VEL
LIN {X 0,Y 270.19,Z 176.322,A -85,B 0,C 180,E1 -17785.092,E2 -17785.092} C_VEL
LIN {X 0,Y 270.176,Z 176.322,A -85,B 0,C 180,E1 -17789.135,E2 -17789.135} C_VEL
LIN {X 0,Y 270.214,Z 176.319,A -85,B 0,C 180,E1 -17792.161,E2 -17792.161} C_VEL
LIN {X 0,Y 270.218,Z 176.322,A -85,B 0,C 180,E1 -17795.541,E2 -17795.541} C_VEL
LIN {X 0,Y 270.214,Z 176.316,A -85,B 0,C 180,E1 -17800.237,E2 -17800.237} C_VEL
LIN {X 0,Y 270.358,Z 176.297,A -85,B 0,C 180,E1 -17804.932,E2 -17804.932} C_VEL
LIN {X 0,Y 270.377,Z 176.298,A -85,B 0,C 180,E1 -17809.516,E2 -17809.516} C_VEL
LIN {X 0,Y 270.559,Z 176.274,A -85,B 0,C 180,E1 -17812.537,E2 -17812.537} C_VEL
LIN {X 0,Y 270.759,Z 176.259,A -85,B 0,C 180,E1 -17818.512,E2 -17818.512} C_VEL
LIN {X 0,Y 270.764,Z 176.258,A -85,B 0,C 180,E1 -17821.487,E2 -17821.487} C_VEL
LIN {X 0,Y 270.562,Z 176.283,A -85,B 0,C 180,E1 -17827.462,E2 -17827.462} C_VEL
LIN {X 0,Y 270.394,Z 176.306,A -85,B 0,C 180,E1 -17830.482,E2 -17830.482} C_VEL
LIN {X 0,Y 270.356,Z 176.31,A -85,B 0,C 180,E1 -17835.067,E2 -17835.067} C_VEL
LIN {X 0,Y 270.28,Z 176.475,A -85,B 0,C 180,E1 -17837.204,E2 -17837.204} C_VEL
LIN {X 0,Y 272.087,Z 183.126,A -85,B 0,C 180,E1 -17840.407,E2 -17840.407} C_VEL
LIN {X 0,Y 272.554,Z 184.449,A -85,B 0,C 180,E1 -17840.765,E2 -17840.765} C_VEL
LIN {X 0,Y 279.382,Z 196.568,A -85,B 0,C 180,E1 -17842.391,E2 -17842.391} C_VEL
LIN {X 0,Y 286.177,Z 210.781,A -85,B 0,C 180,E1 -17843.946,E2 -17843.946} C_VEL
LIN {X 0,Y 289.937,Z 219.822,A -85,B 0,C 180,E1 -17844.788,E2 -17844.788} C_VEL
LIN {X 0,Y 290.597,Z 223.506,A -85,B 0,C 180,E1 -17845,E2 -17845} C_VEL
LIN {X 0,Y 287.588,Z 291.782,A -85,B 0,C 180,E1 -17846.882,E2 -17846.882} C_VEL
LIN {X 0,Y 286.456,Z 304.8,A -85,B 0,C 180,E1 -17847.498,E2 -17847.498} C_VEL
LIN {X 0,Y 285.013,Z 317.213,A -85,B 0,C 180,E1 -17848.362,E2 -17848.362} C_VEL
LIN {X 0,Y 283.143,Z 329.347,A -85,B 0,C 180,E1 -17849.511,E2 -17849.511} C_VEL
LIN {X 0,Y 280.902,Z 341.593,A -85,B 0,C 180,E1 -17851.032,E2 -17851.032} C_VEL
LIN {X 0,Y 278.671,Z 351.97,A -85,B 0,C 180,E1 -17852.683,E2 -17852.683} C_VEL
LIN {X 0,Y 276.353,Z 361.512,A -85,B 0,C 180,E1 -17854.584,E2 -17854.584} C_VEL
LIN {X 0,Y 274.21,Z 370.334,A -85,B 0,C 180,E1 -17856.802,E2 -17856.802} C_VEL
LIN {X 0,Y 272.595,Z 376.395,A -85,B 0,C 180,E1 -17858.7,E2 -17858.7} C_VEL
LIN {X 0,Y 270.914,Z 382.721,A -85,B 0,C 180,E1 -17861.212,E2 -17861.212} C_VEL
LIN {X 0,Y 269.565,Z 388.046,A -85,B 0,C 180,E1 -17864.054,E2 -17864.054} C_VEL
LIN {X 0,Y 268.869,Z 390.856,A -85,B 0,C 180,E1 -17866.161,E2 -17866.161} C_VEL
LIN {X 0,Y 268.181,Z 393.378,A -85,B 0,C 180,E1 -17869.072,E2 -17869.072} C_VEL
LIN {X 0,Y 267.814,Z 394.342,A -85,B 0,C 180,E1 -17871.929,E2 -17871.929} C_VEL
LIN {X 0,Y 267.737,Z 393.909,A -85,B 0,C 180,E1 -17874.728,E2 -17874.728} C_VEL
LIN {X 0,Y 267.839,Z 392.422,A -85,B 0,C 180,E1 -17877.104,E2 -17877.104} C_VEL
LIN {X 0,Y 268.278,Z 389.421,A -85,B 0,C 180,E1 -17879.823,E2 -17879.823} C_VEL
LIN {X 0,Y 268.69,Z 386.117,A -85,B 0,C 180,E1 -17881.915,E2 -17881.915} C_VEL
LIN {X 0,Y 269.465,Z 380.6,A -85,B 0,C 180,E1 -17884.513,E2 -17884.513} C_VEL
LIN {X 0,Y 270.508,Z 373.518,A -85,B 0,C 180,E1 -17887.066,E2 -17887.066} C_VEL
LIN {X 0,Y 271.683,Z 366.088,A -85,B 0,C 180,E1 -17889.174,E2 -17889.174} C_VEL
LIN {X 0,Y 273.094,Z 357.136,A -85,B 0,C 180,E1 -17891.211,E2 -17891.211} C_VEL
LIN {X 0,Y 274.687,Z 346.904,A -85,B 0,C 180,E1 -17893.082,E2 -17893.082} C_VEL
LIN {X 0,Y 276.161,Z 336.822,A -85,B 0,C 180,E1 -17894.557,E2 -17894.557} C_VEL
LIN {X 0,Y 277.602,Z 325.22,A -85,B 0,C 180,E1 -17895.898,E2 -17895.898} C_VEL
LIN {X 0,Y 278.903,Z 312.277,A -85,B 0,C 180,E1 -17897.043,E2 -17897.043} C_VEL
LIN {X 0,Y 279.921,Z 299.621,A -85,B 0,C 180,E1 -17897.835,E2 -17897.835} C_VEL
LIN {X 0,Y 280.663,Z 286.311,A -85,B 0,C 180,E1 -17898.37,E2 -17898.37} C_VEL
LIN {X 0,Y 282.592,Z 219.264,A -85,B 0,C 180,E1 -17900.202,E2 -17900.202} C_VEL
LIN {X 0,Y 280.138,Z 206.113,A -85,B 0,C 180,E1 -17900.799,E2 -17900.799} C_VEL
LIN {X 0,Y 271.996,Z 183.417,A -85,B 0,C 180,E1 -17902.252,E2 -17902.252} C_VEL
LIN {X 0,Y 270.967,Z 178.452,A -85,B 0,C 180,E1 -17904.047,E2 -17904.047} C_VEL
LIN {X 0,Y 270.489,Z 176.333,A -85,B 0,C 180,E1 -17904.971,E2 -17904.971} C_VEL
LIN {X 0,Y 270.785,Z 176.254,A -85,B 0,C 180,E1 -17908.514,E2 -17908.514} C_VEL
LIN {X 0,Y 270.784,Z 176.253,A -85,B 0,C 180,E1 -17911.489,E2 -17911.489} C_VEL
LIN {X 0,Y 270.583,Z 176.277,A -85,B 0,C 180,E1 -17917.463,E2 -17917.463} C_VEL
LIN {X 0,Y 270.408,Z 176.3,A -85,B 0,C 180,E1 -17920.484,E2 -17920.484} C_VEL
LIN {X 0,Y 270.402,Z 176.302,A -85,B 0,C 180,E1 -17925.066,E2 -17925.066} C_VEL
LIN {X 0,Y 270.301,Z 176.311,A -85,B 0,C 180,E1 -17929.757,E2 -17929.757} C_VEL
LIN {X 0,Y 270.274,Z 176.315,A -85,B 0,C 180,E1 -17934.587,E2 -17934.587} C_VEL
LIN {X 0,Y 270.27,Z 176.312,A -85,B 0,C 180,E1 -17937.91,E2 -17937.91} C_VEL
LIN {X 0,Y 270.184,Z 176.33,A -85,B 0,C 180,E1 -17941.349,E2 -17941.349} C_VEL
LIN {X 0,Y 270.202,Z 176.316,A -85,B 0,C 180,E1 -17944.907,E2 -17944.907} C_VEL
LIN {X 0,Y 270.198,Z 176.321,A -85,B 0,C 180,E1 -17948.712,E2 -17948.712} C_VEL
LIN {X 0,Y 270.172,Z 176.329,A -85,B 0,C 180,E1 -17953.252,E2 -17953.252} C_VEL
LIN {X 0,Y 270.175,Z 176.312,A -85,B 0,C 180,E1 -17957.443,E2 -17957.443} C_VEL
LIN {X 0,Y 270.208,Z 176.318,A -85,B 0,C 180,E1 -17961.375,E2 -17961.375} C_VEL
LIN {X 0,Y 270.199,Z 176.327,A -85,B 0,C 180,E1 -17965.095,E2 -17965.095} C_VEL
LIN {X 0,Y 270.186,Z 176.323,A -85,B 0,C 180,E1 -17969.138,E2 -17969.138} C_VEL
LIN {X 0,Y 270.224,Z 176.324,A -85,B 0,C 180,E1 -17972.164,E2 -17972.164} C_VEL
LIN {X 0,Y 270.23,Z 176.319,A -85,B 0,C 180,E1 -17975.543,E2 -17975.543} C_VEL
LIN {X 0,Y 270.304,Z 176.316,A -85,B 0,C 180,E1 -17980.245,E2 -17980.245} C_VEL
LIN {X 0,Y 270.399,Z 176.295,A -85,B 0,C 180,E1 -17984.936,E2 -17984.936} C_VEL
LIN {X 0,Y 270.413,Z 176.3,A -85,B 0,C 180,E1 -17989.519,E2 -17989.519} C_VEL
LIN {X 0,Y 270.524,Z 176.279,A -85,B 0,C 180,E1 -17991.759,E2 -17991.759} C_VEL
LIN {X 0,Y 269.861,Z 176.364,A -85,B 0,C 180,E1 -17993,E2 -17993} C_VEL
LIN {X 0,Y 266.978,Z 176.726,A -85,B 0,C 180,E1 -17995.022,E2 -17995.022} C_VEL
LIN {X 0,Y 264.612,Z 177.022,A -85,B 0,C 180,E1 -17996.666,E2 -17996.666} C_VEL
LIN {X 0,Y 263.724,Z 177.133,A -85,B 0,C 180,E1 -17997.941,E2 -17997.941} C_VEL
LIN {X 0,Y 263.72,Z 177.129,A -85,B 0,C 180,E1 -17998.371,E2 -17998.371} C_VEL
LIN {X 0,Y 263.737,Z 177.117,A -85,B 0,C 180,E1 -18001.528,E2 -18001.528} C_VEL
LIN {X 0,Y 263.528,Z 177.156,A -85,B 0,C 180,E1 -18007.664,E2 -18007.664} C_VEL
LIN {X 0,Y 263.353,Z 177.179,A -85,B 0,C 180,E1 -18010.767,E2 -18010.767} C_VEL
LIN {X 0,Y 263.314,Z 177.168,A -85,B 0,C 180,E1 -18015.481,E2 -18015.481} C_VEL
LIN {X 0,Y 263.212,Z 177.196,A -85,B 0,C 180,E1 -18020.311,E2 -18020.311} C_VEL
LIN {X 0,Y 263.129,Z 177.196,A -85,B 0,C 180,E1 -18025.3,E2 -18025.3} C_VEL
LIN {X 0,Y 263.133,Z 177.205,A -85,B 0,C 180,E1 -18028.736,E2 -18028.736} C_VEL
LIN {X 0,Y 263.132,Z 177.204,A -85,B 0,C 180,E1 -18032.289,E2 -18032.289} C_VEL
LIN {X 0,Y 263.18,Z 177.202,A -85,B 0,C 180,E1 -18036.761,E2 -18036.761} C_VEL
LIN {X 0,Y 263.096,Z 177.204,A -85,B 0,C 180,E1 -18039.875,E2 -18039.875} C_VEL
LIN {X 0,Y 263.081,Z 177.212,A -85,B 0,C 180,E1 -18043.994,E2 -18043.994} C_VEL
LIN {X 0,Y 263.079,Z 177.214,A -85,B 0,C 180,E1 -18048.097,E2 -18048.097} C_VEL
LIN {X 0,Y 263.108,Z 177.211,A -85,B 0,C 180,E1 -18052.093,E2 -18052.093} C_VEL
LIN {X 0,Y 263.165,Z 177.261,A -85,B 0,C 180,E1 -18056.018,E2 -18056.018} C_VEL
LIN {X 0,Y 264.369,Z 182.92,A -85,B 0,C 180,E1 -18058.288,E2 -18058.288} C_VEL
LIN {X 0,Y 266.059,Z 190.945,A -85,B 0,C 180,E1 -18061.21,E2 -18061.21} C_VEL
LIN {X 0,Y 268.999,Z 199.256,A -85,B 0,C 180,E1 -18061.805,E2 -18061.805} C_VEL
LIN {X 0,Y 271.783,Z 207.596,A -85,B 0,C 180,E1 -18062.315,E2 -18062.315} C_VEL
LIN {X 0,Y 275.807,Z 234.73,A -85,B 0,C 180,E1 -18063.494,E2 -18063.494} C_VEL
LIN {X 0,Y 273.696,Z 299.66,A -85,B 0,C 180,E1 -18065.336,E2 -18065.336} C_VEL
LIN {X 0,Y 272.664,Z 313.791,A -85,B 0,C 180,E1 -18066.047,E2 -18066.047} C_VEL
LIN {X 0,Y 271.473,Z 325.857,A -85,B 0,C 180,E1 -18066.947,E2 -18066.947} C_VEL
LIN {X 0,Y 269.852,Z 338.399,A -85,B 0,C 180,E1 -18068.214,E2 -18068.214} C_VEL
LIN {X 0,Y 268.288,Z 349.654,A -85,B 0,C 180,E1 -18069.689,E2 -18069.689} C_VEL
LIN {X 0,Y 266.868,Z 358.768,A -85,B 0,C 180,E1 -18071.178,E2 -18071.178} C_VEL
LIN {X 0,Y 265.488,Z 368.126,A -85,B 0,C 180,E1 -18073.069,E2 -18073.069} C_VEL
LIN {X 0,Y 263.913,Z 377.189,A -85,B 0,C 180,E1 -18075.344,E2 -18075.344} C_VEL
LIN {X 0,Y 262.682,Z 384.466,A -85,B 0,C 180,E1 -18077.639,E2 -18077.639} C_VEL
LIN {X 0,Y 261.899,Z 390.251,A -85,B 0,C 180,E1 -18079.953,E2 -18079.953} C_VEL
LIN {X 0,Y 261.365,Z 394.782,A -85,B 0,C 180,E1 -18082.272,E2 -18082.272} C_VEL
LIN {X 0,Y 261.088,Z 398.514,A -85,B 0,C 180,E1 -18084.861,E2 -18084.861} C_VEL
LIN {X 0,Y 261.028,Z 400.597,A -85,B 0,C 180,E1 -18086.912,E2 -18086.912} C_VEL
LIN {X 0,Y 261.039,Z 401.635,A -85,B 0,C 180,E1 -18088.456,E2 -18088.456} C_VEL
LIN {X 0,Y 261.084,Z 402.275,A -85,B 0,C 180,E1 -18089.998,E2 -18089.998} C_VEL
LIN {X 0,Y 261.038,Z 402.519,A -85,B 0,C 180,E1 -18091.541,E2 -18091.541} C_VEL
LIN {X 0,Y 261.018,Z 402.347,A -85,B 0,C 180,E1 -18093.085,E2 -18093.085} C_VEL
LIN {X 0,Y 261.236,Z 400.766,A -85,B 0,C 180,E1 -18096.176,E2 -18096.176} C_VEL
LIN {X 0,Y 261.504,Z 399.386,A -85,B 0,C 180,E1 -18097.721,E2 -18097.721} C_VEL
LIN {X 0,Y 262.111,Z 396.483,A -85,B 0,C 180,E1 -18100.035,E2 -18100.035} C_VEL
LIN {X 0,Y 263.063,Z 392.556,A -85,B 0,C 180,E1 -18102.339,E2 -18102.339} C_VEL
LIN {X 0,Y 264.321,Z 387.509,A -85,B 0,C 180,E1 -18104.629,E2 -18104.629} C_VEL
LIN {X 0,Y 266.193,Z 381.186,A -85,B 0,C 180,E1 -18106.881,E2 -18106.881} C_VEL
LIN {X 0,Y 267.856,Z 374.726,A -85,B 0,C 180,E1 -18108.757,E2 -18108.757} C_VEL
LIN {X 0,Y 269.743,Z 367.084,A -85,B 0,C 180,E1 -18110.591,E2 -18110.591} C_VEL
LIN {X 0,Y 272.253,Z 356.698,A -85,B 0,C 180,E1 -18112.579,E2 -18112.579} C_VEL
LIN {X 0,Y 274.608,Z 346.171,A -85,B 0,C 180,E1 -18114.17,E2 -18114.17} C_VEL
LIN {X 0,Y 276.912,Z 334.448,A -85,B 0,C 180,E1 -18115.558,E2 -18115.558} C_VEL
LIN {X 0,Y 278.889,Z 322.036,A -85,B 0,C 180,E1 -18116.669,E2 -18116.669} C_VEL
LIN {X 0,Y 280.503,Z 309.124,A -85,B 0,C 180,E1 -18117.511,E2 -18117.511} C_VEL
LIN {X 0,Y 281.532,Z 296.482,A -85,B 0,C 180,E1 -18118.058,E2 -18118.058} C_VEL
LIN {X 0,Y 284.173,Z 236.963,A -85,B 0,C 180,E1 -18119.726,E2 -18119.726} C_VEL
LIN {X 0,Y 281.942,Z 222.519,A -85,B 0,C 180,E1 -18120.559,E2 -18120.559} C_VEL
LIN {X 0,Y 281.132,Z 219.483,A -85,B 0,C 180,E1 -18120.79,E2 -18120.79} C_VEL
LIN {X 0,Y 275.012,Z 205.822,A -85,B 0,C 180,E1 -18122.267,E2 -18122.267} C_VEL
LIN {X 0,Y 268.811,Z 193.996,A -85,B 0,C 180,E1 -18123.803,E2 -18123.803} C_VEL
LIN {X 0,Y 266.604,Z 189.673,A -85,B 0,C 180,E1 -18124.467,E2 -18124.467} C_VEL
LIN {X 0,Y 264.715,Z 182.811,A -85,B 0,C 180,E1 -18127.633,E2 -18127.633} C_VEL
LIN {X 0,Y 263.111,Z 177.249,A -85,B 0,C 180,E1 -18130.589,E2 -18130.589} C_VEL
LIN {X 0,Y 263.07,Z 177.214,A -85,B 0,C 180,E1 -18133.992,E2 -18133.992} C_VEL
LIN {X 0,Y 263.102,Z 177.212,A -85,B 0,C 180,E1 -18138.409,E2 -18138.409} C_VEL
LIN {X 0,Y 263.132,Z 177.201,A -85,B 0,C 180,E1 -18142.098,E2 -18142.098} C_VEL
LIN {X 0,Y 263.144,Z 177.199,A -85,B 0,C 180,E1 -18145.884,E2 -18145.884} C_VEL
LIN {X 0,Y 263.115,Z 177.202,A -85,B 0,C 180,E1 -18149.502,E2 -18149.502} C_VEL
LIN {X 0,Y 263.132,Z 177.199,A -85,B 0,C 180,E1 -18152.995,E2 -18152.995} C_VEL
LIN {X 0,Y 263.134,Z 177.198,A -85,B 0,C 180,E1 -18156.382,E2 -18156.382} C_VEL
LIN {X 0,Y 263.199,Z 177.194,A -85,B 0,C 180,E1 -18159.688,E2 -18159.688} C_VEL
LIN {X 0,Y 263.3,Z 177.176,A -85,B 0,C 180,E1 -18164.518,E2 -18164.518} C_VEL
LIN {X 0,Y 263.323,Z 177.174,A -85,B 0,C 180,E1 -18169.232,E2 -18169.232} C_VEL
LIN {X 0,Y 263.521,Z 177.151,A -85,B 0,C 180,E1 -18172.336,E2 -18172.336} C_VEL
LIN {X 0,Y 263.723,Z 177.136,A -85,B 0,C 180,E1 -18178.472,E2 -18178.472} C_VEL
LIN {X 0,Y 263.727,Z 177.134,A -85,B 0,C 180,E1 -18181.526,E2 -18181.526} C_VEL
LIN {X 0,Y 263.524,Z 177.161,A -85,B 0,C 180,E1 -18187.662,E2 -18187.662} C_VEL
LIN {X 0,Y 263.334,Z 177.184,A -85,B 0,C 180,E1 -18190.767,E2 -18190.767} C_VEL
LIN {X 0,Y 263.298,Z 177.187,A -85,B 0,C 180,E1 -18195.48,E2 -18195.48} C_VEL
LIN {X 0,Y 263.294,Z 177.46,A -85,B 0,C 180,E1 -18196.077,E2 -18196.077} C_VEL
LIN {X 0,Y 265.099,Z 183.964,A -85,B 0,C 180,E1 -18199.302,E2 -18199.302} C_VEL
LIN {X 0,Y 270.683,Z 193.75,A -85,B 0,C 180,E1 -18200.808,E2 -18200.808} C_VEL
LIN {X 0,Y 275.871,Z 203.44,A -85,B 0,C 180,E1 -18202.072,E2 -18202.072} C_VEL
LIN {X 0,Y 282.458,Z 217.718,A -85,B 0,C 180,E1 -18203.629,E2 -18203.629} C_VEL
LIN {X 0,Y 284.499,Z 223.231,A -85,B 0,C 180,E1 -18204.127,E2 -18204.127} C_VEL
LIN {X 0,Y 284.686,Z 226.437,A -85,B 0,C 180,E1 -18204.265,E2 -18204.265} C_VEL
LIN {X 0,Y 281.626,Z 291.938,A -85,B 0,C 180,E1 -18206.11,E2 -18206.11} C_VEL
LIN {X 0,Y 280.427,Z 305.162,A -85,B 0,C 180,E1 -18206.749,E2 -18206.749} C_VEL
LIN {X 0,Y 278.921,Z 317.452,A -85,B 0,C 180,E1 -18207.622,E2 -18207.622} C_VEL
LIN {X 0,Y 276.911,Z 329.904,A -85,B 0,C 180,E1 -18208.83,E2 -18208.83} C_VEL
LIN {X 0,Y 274.71,Z 341.294,A -85,B 0,C 180,E1 -18210.268,E2 -18210.268} C_VEL
LIN {X 0,Y 272.688,Z 350.555,A -85,B 0,C 180,E1 -18211.737,E2 -18211.737} C_VEL
LIN {X 0,Y 270.2,Z 360.368,A -85,B 0,C 180,E1 -18213.665,E2 -18213.665} C_VEL
LIN {X 0,Y 268.149,Z 368.437,A -85,B 0,C 180,E1 -18215.664,E2 -18215.664} C_VEL
LIN {X 0,Y 266.27,Z 374.983,A -85,B 0,C 180,E1 -18217.647,E2 -18217.647} C_VEL
LIN {X 0,Y 264.438,Z 381.596,A -85,B 0,C 180,E1 -18220.177,E2 -18220.177} C_VEL
LIN {X 0,Y 263.005,Z 386.751,A -85,B 0,C 180,E1 -18222.781,E2 -18222.781} C_VEL
LIN {X 0,Y 261.884,Z 390.902,A -85,B 0,C 180,E1 -18225.757,E2 -18225.757} C_VEL
LIN {X 0,Y 261.107,Z 393.545,A -85,B 0,C 180,E1 -18228.907,E2 -18228.907} C_VEL
LIN {X 0,Y 260.741,Z 394.451,A -85,B 0,C 180,E1 -18231.691,E2 -18231.691} C_VEL
LIN {X 0,Y 260.621,Z 394.224,A -85,B 0,C 180,E1 -18233.996,E2 -18233.996} C_VEL
LIN {X 0,Y 260.697,Z 392.811,A -85,B 0,C 180,E1 -18236.689,E2 -18236.689} C_VEL
LIN {X 0,Y 261.098,Z 390.037,A -85,B 0,C 180,E1 -18239.466,E2 -18239.466} C_VEL
LIN {X 0,Y 261.552,Z 386.59,A -85,B 0,C 180,E1 -18241.787,E2 -18241.787} C_VEL
LIN {X 0,Y 262.389,Z 380.818,A -85,B 0,C 180,E1 -18244.626,E2 -18244.626} C_VEL
LIN {X 0,Y 263.47,Z 373.756,A -85,B 0,C 180,E1 -18247.248,E2 -18247.248} C_VEL
LIN {X 0,Y 264.708,Z 366.247,A -85,B 0,C 180,E1 -18249.44,E2 -18249.44} C_VEL
LIN {X 0,Y 266.164,Z 357.304,A -85,B 0,C 180,E1 -18251.529,E2 -18251.529} C_VEL
LIN {X 0,Y 267.783,Z 347.244,A -85,B 0,C 180,E1 -18253.418,E2 -18253.418} C_VEL
LIN {X 0,Y 269.433,Z 336.265,A -85,B 0,C 180,E1 -18255.054,E2 -18255.054} C_VEL
LIN {X 0,Y 271.005,Z 323.75,A -85,B 0,C 180,E1 -18256.505,E2 -18256.505} C_VEL
LIN {X 0,Y 272.167,Z 312.396,A -85,B 0,C 180,E1 -18257.512,E2 -18257.512} C_VEL
LIN {X 0,Y 273.278,Z 299.179,A -85,B 0,C 180,E1 -18258.349,E2 -18258.349} C_VEL
LIN {X 0,Y 274.031,Z 285.25,A -85,B 0,C 180,E1 -18258.909,E2 -18258.909} C_VEL
LIN {X 0,Y 276.068,Z 220.631,A -85,B 0,C 180,E1 -18260.703,E2 -18260.703} C_VEL
LIN {X 0,Y 273.769,Z 208.191,A -85,B 0,C 180,E1 -18261.281,E2 -18261.281} C_VEL
LIN {X 0,Y 264.88,Z 183.681,A -85,B 0,C 180,E1 -18262.905,E2 -18262.905} C_VEL
LIN {X 0,Y 264.668,Z 182.764,A -85,B 0,C 180,E1 -18263.139,E2 -18263.139} C_VEL
LIN {X 0,Y 263.396,Z 177.233,A -85,B 0,C 180,E1 -18265.41,E2 -18265.41} C_VEL
LIN {X 0,Y 263.749,Z 177.13,A -85,B 0,C 180,E1 -18268.475,E2 -18268.475} C_VEL
LIN {X 0,Y 263.748,Z 177.129,A -85,B 0,C 180,E1 -18271.528,E2 -18271.528} C_VEL
LIN {X 0,Y 263.542,Z 177.153,A -85,B 0,C 180,E1 -18277.664,E2 -18277.664} C_VEL
LIN {X 0,Y 263.348,Z 177.18,A -85,B 0,C 180,E1 -18280.768,E2 -18280.768} C_VEL
LIN {X 0,Y 263.35,Z 177.183,A -85,B 0,C 180,E1 -18285.479,E2 -18285.479} C_VEL
LIN {X 0,Y 263.263,Z 177.186,A -85,B 0,C 180,E1 -18290.308,E2 -18290.308} C_VEL
LIN {X 0,Y 263.208,Z 177.189,A -85,B 0,C 180,E1 -18295.293,E2 -18295.293} C_VEL
LIN {X 0,Y 263.165,Z 177.199,A -85,B 0,C 180,E1 -18298.733,E2 -18298.733} C_VEL
LIN {X 0,Y 263.133,Z 177.206,A -85,B 0,C 180,E1 -18302.29,E2 -18302.29} C_VEL
LIN {X 0,Y 263.182,Z 177.185,A -85,B 0,C 180,E1 -18306.764,E2 -18306.764} C_VEL
LIN {X 0,Y 263.126,Z 177.207,A -85,B 0,C 180,E1 -18311.595,E2 -18311.595} C_VEL
LIN {X 0,Y 263.129,Z 177.199,A -85,B 0,C 180,E1 -18316.018,E2 -18316.018} C_VEL
LIN {X 0,Y 263.106,Z 177.194,A -85,B 0,C 180,E1 -18320.129,E2 -18320.129} C_VEL
LIN {X 0,Y 263.159,Z 177.202,A -85,B 0,C 180,E1 -18324.018,E2 -18324.018} C_VEL
LIN {X 0,Y 263.129,Z 177.204,A -85,B 0,C 180,E1 -18327.712,E2 -18327.712} C_VEL
LIN {X 0,Y 263.15,Z 177.204,A -85,B 0,C 180,E1 -18331.806,E2 -18331.806} C_VEL
LIN {X 0,Y 263.192,Z 177.196,A -85,B 0,C 180,E1 -18335.219,E2 -18335.219} C_VEL
LIN {X 0,Y 263.265,Z 177.189,A -85,B 0,C 180,E1 -18339.694,E2 -18339.694} C_VEL
LIN {X 0,Y 263.348,Z 177.174,A -85,B 0,C 180,E1 -18344.523,E2 -18344.523} C_VEL
LIN {X 0,Y 263.355,Z 177.178,A -85,B 0,C 180,E1 -18349.234,E2 -18349.234} C_VEL
LIN {X 0,Y 263.528,Z 177.153,A -85,B 0,C 180,E1 -18352.338,E2 -18352.338} C_VEL
LIN {X 0,Y 263.72,Z 177.129,A -85,B 0,C 180,E1 -18358.371,E2 -18358.371} C_VEL
LIN {X 0,Y 263.513,Z 177.158,A -85,B 0,C 180,E1 -18359.223,E2 -18359.223} C_VEL
LIN {X 0,Y 262.715,Z 177.257,A -85,B 0,C 180,E1 -18360.062,E2 -18360.062} C_VEL
LIN {X 0,Y 258.738,Z 177.742,A -85,B 0,C 180,E1 -18362.546,E2 -18362.546} C_VEL
LIN {X 0,Y 256.628,Z 177.999,A -85,B 0,C 180,E1 -18364.268,E2 -18364.268} C_VEL
LIN {X 0,Y 256.329,Z 178.037,A -85,B 0,C 180,E1 -18365.157,E2 -18365.157} C_VEL
LIN {X 0,Y 256.492,Z 178.034,A -85,B 0,C 180,E1 -18367.875,E2 -18367.875} C_VEL
LIN {X 0,Y 256.294,Z 178.059,A -85,B 0,C 180,E1 -18371.067,E2 -18371.067} C_VEL
LIN {X 0,Y 256.234,Z 178.048,A -85,B 0,C 180,E1 -18375.92,E2 -18375.92} C_VEL
LIN {X 0,Y 256.123,Z 178.082,A -85,B 0,C 180,E1 -18381.097,E2 -18381.097} C_VEL
LIN {X 0,Y 256.089,Z 178.074,A -85,B 0,C 180,E1 -18385.089,E2 -18385.089} C_VEL
LIN {X 0,Y 256.091,Z 178.081,A -85,B 0,C 180,E1 -18388.574,E2 -18388.574} C_VEL
LIN {X 0,Y 256.078,Z 178.083,A -85,B 0,C 180,E1 -18391.701,E2 -18391.701} C_VEL
LIN {X 0,Y 256.084,Z 178.081,A -85,B 0,C 180,E1 -18395.193,E2 -18395.193} C_VEL
LIN {X 0,Y 256.114,Z 178.083,A -85,B 0,C 180,E1 -18397.269,E2 -18397.269} C_VEL
LIN {X 0,Y 256.023,Z 178.091,A -85,B 0,C 180,E1 -18401.211,E2 -18401.211} C_VEL
LIN {X 0,Y 256.022,Z 178.089,A -85,B 0,C 180,E1 -18405.539,E2 -18405.539} C_VEL
LIN {X 0,Y 256.013,Z 178.094,A -85,B 0,C 180,E1 -18408.787,E2 -18408.787} C_VEL
LIN {X 0,Y 256.104,Z 178.083,A -85,B 0,C 180,E1 -18412.862,E2 -18412.862} C_VEL
LIN {X 0,Y 256.125,Z 178.167,A -85,B 0,C 180,E1 -18415.558,E2 -18415.558} C_VEL
LIN {X 0,Y 258.317,Z 188.588,A -85,B 0,C 180,E1 -18419.718,E2 -18419.718} C_VEL
LIN {X 0,Y 258.884,Z 191.081,A -85,B 0,C 180,E1 -18420.538,E2 -18420.538} C_VEL
LIN {X 0,Y 265.242,Z 208.772,A -85,B 0,C 180,E1 -18421.766,E2 -18421.766} C_VEL
LIN {X 0,Y 269.182,Z 235.602,A -85,B 0,C 180,E1 -18422.968,E2 -18422.968} C_VEL
LIN {X 0,Y 267,Z 299.643,A -85,B 0,C 180,E1 -18424.831,E2 -18424.831} C_VEL
LIN {X 0,Y 265.95,Z 313.74,A -85,B 0,C 180,E1 -18425.559,E2 -18425.559} C_VEL
LIN {X 0,Y 264.653,Z 326.277,A -85,B 0,C 180,E1 -18426.525,E2 -18426.525} C_VEL
LIN {X 0,Y 263.004,Z 338.716,A -85,B 0,C 180,E1 -18427.823,E2 -18427.823} C_VEL
LIN {X 0,Y 261.396,Z 349.887,A -85,B 0,C 180,E1 -18429.335,E2 -18429.335} C_VEL
LIN {X 0,Y 259.764,Z 359.933,A -85,B 0,C 180,E1 -18431.053,E2 -18431.053} C_VEL
LIN {X 0,Y 258.355,Z 369.067,A -85,B 0,C 180,E1 -18432.995,E2 -18432.995} C_VEL
LIN {X 0,Y 256.757,Z 377.953,A -85,B 0,C 180,E1 -18435.332,E2 -18435.332} C_VEL
LIN {X 0,Y 255.56,Z 385.023,A -85,B 0,C 180,E1 -18437.693,E2 -18437.693} C_VEL
LIN {X 0,Y 254.661,Z 391.489,A -85,B 0,C 180,E1 -18440.467,E2 -18440.467} C_VEL
LIN {X 0,Y 254.178,Z 395.709,A -85,B 0,C 180,E1 -18442.851,E2 -18442.851} C_VEL
LIN {X 0,Y 253.977,Z 398.834,A -85,B 0,C 180,E1 -18445.236,E2 -18445.236} C_VEL
LIN {X 0,Y 253.931,Z 400.376,A -85,B 0,C 180,E1 -18446.825,E2 -18446.825} C_VEL
LIN {X 0,Y 253.949,Z 401.453,A -85,B 0,C 180,E1 -18448.413,E2 -18448.413} C_VEL
LIN {X 0,Y 254.012,Z 402.121,A -85,B 0,C 180,E1 -18449.998,E2 -18449.998} C_VEL
LIN {X 0,Y 253.948,Z 402.393,A -85,B 0,C 180,E1 -18451.584,E2 -18451.584} C_VEL
LIN {X 0,Y 253.922,Z 402.269,A -85,B 0,C 180,E1 -18453.172,E2 -18453.172} C_VEL
LIN {X 0,Y 254.023,Z 401.521,A -85,B 0,C 180,E1 -18455.117,E2 -18455.117} C_VEL
LIN {X 0,Y 254.441,Z 399.397,A -85,B 0,C 180,E1 -18457.937,E2 -18457.937} C_VEL
LIN {X 0,Y 255.106,Z 396.551,A -85,B 0,C 180,E1 -18460.314,E2 -18460.314} C_VEL
LIN {X 0,Y 256.108,Z 392.697,A -85,B 0,C 180,E1 -18462.68,E2 -18462.68} C_VEL
LIN {X 0,Y 257.455,Z 387.732,A -85,B 0,C 180,E1 -18465.028,E2 -18465.028} C_VEL
LIN {X 0,Y 259.428,Z 381.5,A -85,B 0,C 180,E1 -18467.335,E2 -18467.335} C_VEL
LIN {X 0,Y 261.082,Z 375.325,A -85,B 0,C 180,E1 -18469.203,E2 -18469.203} C_VEL
LIN {X 0,Y 263.125,Z 367.582,A -85,B 0,C 180,E1 -18471.134,E2 -18471.134} C_VEL
LIN {X 0,Y 265.53,Z 358.424,A -85,B 0,C 180,E1 -18472.977,E2 -18472.977} C_VEL
LIN {X 0,Y 267.888,Z 348.291,A -85,B 0,C 180,E1 -18474.61,E2 -18474.61} C_VEL
LIN {X 0,Y 270.265,Z 337.124,A -85,B 0,C 180,E1 -18476.026,E2 -18476.026} C_VEL
LIN {X 0,Y 272.501,Z 324.7,A -85,B 0,C 180,E1 -18477.242,E2 -18477.242} C_VEL
LIN {X 0,Y 274.267,Z 312.052,A -85,B 0,C 180,E1 -18478.139,E2 -18478.139} C_VEL
LIN {X 0,Y 275.484,Z 299.043,A -85,B 0,C 180,E1 -18478.783,E2 -18478.783} C_VEL
LIN {X 0,Y 278.432,Z 239.005,A -85,B 0,C 180,E1 -18480.51,E2 -18480.51} C_VEL
LIN {X 0,Y 276.884,Z 227.724,A -85,B 0,C 180,E1 -18481.156,E2 -18481.156} C_VEL
LIN {X 0,Y 275.865,Z 222.79,A -85,B 0,C 180,E1 -18481.497,E2 -18481.497} C_VEL
LIN {X 0,Y 269.595,Z 208.712,A -85,B 0,C 180,E1 -18483.091,E2 -18483.091} C_VEL
LIN {X 0,Y 264.178,Z 198.312,A -85,B 0,C 180,E1 -18484.513,E2 -18484.513} C_VEL
LIN {X 0,Y 260.962,Z 192.72,A -85,B 0,C 180,E1 -18485.401,E2 -18485.401} C_VEL
LIN {X 0,Y 259.339,Z 189.546,A -85,B 0,C 180,E1 -18485.932,E2 -18485.932} C_VEL
LIN {X 0,Y 257.397,Z 182.684,A -85,B 0,C 180,E1 -18489.305,E2 -18489.305} C_VEL
LIN {X 0,Y 256.051,Z 178.129,A -85,B 0,C 180,E1 -18491.944,E2 -18491.944} C_VEL
LIN {X 0,Y 256.022,Z 178.09,A -85,B 0,C 180,E1 -18496.664,E2 -18496.664} C_VEL
LIN {X 0,Y 256.059,Z 178.091,A -85,B 0,C 180,E1 -18500.855,E2 -18500.855} C_VEL
LIN {X 0,Y 256.072,Z 178.082,A -85,B 0,C 180,E1 -18504.805,E2 -18504.805} C_VEL
LIN {X 0,Y 256.074,Z 178.079,A -85,B 0,C 180,E1 -18508.569,E2 -18508.569} C_VEL
LIN {X 0,Y 256.083,Z 178.078,A -85,B 0,C 180,E1 -18512.189,E2 -18512.189} C_VEL
LIN {X 0,Y 256.123,Z 178.076,A -85,B 0,C 180,E1 -18515.694,E2 -18515.694} C_VEL
LIN {X 0,Y 256.115,Z 178.08,A -85,B 0,C 180,E1 -18519.1,E2 -18519.1} C_VEL
LIN {X 0,Y 256.22,Z 178.059,A -85,B 0,C 180,E1 -18524.079,E2 -18524.079} C_VEL
LIN {X 0,Y 256.269,Z 178.052,A -85,B 0,C 180,E1 -18528.932,E2 -18528.932} C_VEL
LIN {X 0,Y 256.484,Z 178.028,A -85,B 0,C 180,E1 -18532.125,E2 -18532.125} C_VEL
LIN {X 0,Y 256.446,Z 178.032,A -85,B 0,C 180,E1 -18536.857,E2 -18536.857} C_VEL
LIN {X 0,Y 256.686,Z 178.012,A -85,B 0,C 180,E1 -18538.43,E2 -18538.43} C_VEL
LIN {X 0,Y 256.689,Z 178.011,A -85,B 0,C 180,E1 -18541.568,E2 -18541.568} C_VEL
LIN {X 0,Y 256.441,Z 178.036,A -85,B 0,C 180,E1 -18546.772,E2 -18546.772} C_VEL
LIN {X 0,Y 256.391,Z 178.043,A -85,B 0,C 180,E1 -18549.466,E2 -18549.466} C_VEL
LIN {X 0,Y 256.242,Z 178.164,A -85,B 0,C 180,E1 -18554.594,E2 -18554.594} C_VEL
LIN {X 0,Y 257.804,Z 183.729,A -85,B 0,C 180,E1 -18557.654,E2 -18557.654} C_VEL
LIN {X 0,Y 258.265,Z 184.925,A -85,B 0,C 180,E1 -18557.966,E2 -18557.966} C_VEL
LIN {X 0,Y 261.859,Z 190.887,A -85,B 0,C 180,E1 -18558.99,E2 -18558.99} C_VEL
LIN {X 0,Y 268.527,Z 202.585,A -85,B 0,C 180,E1 -18560.758,E2 -18560.758} C_VEL
LIN {X 0,Y 274.738,Z 215.452,A -85,B 0,C 180,E1 -18562.332,E2 -18562.332} C_VEL
LIN {X 0,Y 278.915,Z 225.44,A -85,B 0,C 180,E1 -18563.358,E2 -18563.358} C_VEL
LIN {X 0,Y 275.89,Z 290.671,A -85,B 0,C 180,E1 -18565.239,E2 -18565.239} C_VEL
LIN {X 0,Y 274.599,Z 304.116,A -85,B 0,C 180,E1 -18565.867,E2 -18565.867} C_VEL
LIN {X 0,Y 273.118,Z 316.35,A -85,B 0,C 180,E1 -18566.736,E2 -18566.736} C_VEL
LIN {X 0,Y 271.255,Z 327.661,A -85,B 0,C 180,E1 -18567.798,E2 -18567.798} C_VEL
LIN {X 0,Y 268.886,Z 339.61,A -85,B 0,C 180,E1 -18569.275,E2 -18569.275} C_VEL
LIN {X 0,Y 266.421,Z 350.453,A -85,B 0,C 180,E1 -18570.987,E2 -18570.987} C_VEL
LIN {X 0,Y 263.814,Z 360.318,A -85,B 0,C 180,E1 -18572.953,E2 -18572.953} C_VEL
LIN {X 0,Y 261.642,Z 368.411,A -85,B 0,C 180,E1 -18574.993,E2 -18574.993} C_VEL
LIN {X 0,Y 259.454,Z 375.642,A -85,B 0,C 180,E1 -18577.248,E2 -18577.248} C_VEL
LIN {X 0,Y 257.804,Z 381.185,A -85,B 0,C 180,E1 -18579.424,E2 -18579.424} C_VEL
LIN {X 0,Y 256.171,Z 386.677,A -85,B 0,C 180,E1 -18582.209,E2 -18582.209} C_VEL
LIN {X 0,Y 255.268,Z 389.726,A -85,B 0,C 180,E1 -18584.292,E2 -18584.292} C_VEL
LIN {X 0,Y 254.614,Z 391.993,A -85,B 0,C 180,E1 -18586.368,E2 -18586.368} C_VEL
LIN {X 0,Y 254.104,Z 393.552,A -85,B 0,C 180,E1 -18588.413,E2 -18588.413} C_VEL
LIN {X 0,Y 253.719,Z 394.501,A -85,B 0,C 180,E1 -18590.858,E2 -18590.858} C_VEL
LIN {X 0,Y 253.544,Z 394.451,A -85,B 0,C 180,E1 -18593.498,E2 -18593.498} C_VEL
LIN {X 0,Y 253.565,Z 393.132,A -85,B 0,C 180,E1 -18596.338,E2 -18596.338} C_VEL
LIN {X 0,Y 253.913,Z 390.59,A -85,B 0,C 180,E1 -18599.096,E2 -18599.096} C_VEL
LIN {X 0,Y 254.522,Z 386.35,A -85,B 0,C 180,E1 -18602.078,E2 -18602.078} C_VEL
LIN {X 0,Y 255.272,Z 381.375,A -85,B 0,C 180,E1 -18604.588,E2 -18604.588} C_VEL
LIN {X 0,Y 256.224,Z 375.246,A -85,B 0,C 180,E1 -18606.994,E2 -18606.994} C_VEL
LIN {X 0,Y 257.406,Z 368.18,A -85,B 0,C 180,E1 -18609.212,E2 -18609.212} C_VEL
LIN {X 0,Y 258.889,Z 359.577,A -85,B 0,C 180,E1 -18611.391,E2 -18611.391} C_VEL
LIN {X 0,Y 260.512,Z 349.928,A -85,B 0,C 180,E1 -18613.345,E2 -18613.345} C_VEL
LIN {X 0,Y 262.33,Z 338.397,A -85,B 0,C 180,E1 -18615.194,E2 -18615.194} C_VEL
LIN {X 0,Y 263.786,Z 327.949,A -85,B 0,C 180,E1 -18616.521,E2 -18616.521} C_VEL
LIN {X 0,Y 265.073,Z 316.515,A -85,B 0,C 180,E1 -18617.659,E2 -18617.659} C_VEL
LIN {X 0,Y 266.231,Z 303.189,A -85,B 0,C 180,E1 -18618.634,E2 -18618.634} C_VEL
LIN {X 0,Y 267.161,Z 290.345,A -85,B 0,C 180,E1 -18619.256,E2 -18619.256} C_VEL
LIN {X 0,Y 269.412,Z 221.219,A -85,B 0,C 180,E1 -18621.255,E2 -18621.255} C_VEL
LIN {X 0,Y 267.506,Z 210.617,A -85,B 0,C 180,E1 -18621.76,E2 -18621.76} C_VEL
LIN {X 0,Y 258.55,Z 186.113,A -85,B 0,C 180,E1 -18623.405,E2 -18623.405} C_VEL
LIN {X 0,Y 257.564,Z 183.362,A -85,B 0,C 180,E1 -18623.687,E2 -18623.687} C_VEL
LIN {X 0,Y 256.404,Z 178.113,A -85,B 0,C 180,E1 -18625.876,E2 -18625.876} C_VEL
LIN {X 0,Y 256.712,Z 178.007,A -85,B 0,C 180,E1 -18628.433,E2 -18628.433} C_VEL
LIN {X 0,Y 256.711,Z 178.006,A -85,B 0,C 180,E1 -18631.57,E2 -18631.57} C_VEL
LIN {X 0,Y 256.473,Z 178.037,A -85,B 0,C 180,E1 -18636.294,E2 -18636.294} C_VEL
LIN {X 0,Y 256.425,Z 178.042,A -85,B 0,C 180,E1 -18639.467,E2 -18639.467} C_VEL
LIN {X 0,Y 256.254,Z 178.062,A -85,B 0,C 180,E1 -18644.292,E2 -18644.292} C_VEL
LIN {X 0,Y 256.21,Z 178.064,A -85,B 0,C 180,E1 -18647.563,E2 -18647.563} C_VEL
LIN {X 0,Y 256.157,Z 178.075,A -85,B 0,C 180,E1 -18651.121,E2 -18651.121} C_VEL
LIN {X 0,Y 256.188,Z 178.064,A -85,B 0,C 180,E1 -18655.14,E2 -18655.14} C_VEL
LIN {X 0,Y 256.104,Z 178.083,A -85,B 0,C 180,E1 -18659.602,E2 -18659.602} C_VEL
LIN {X 0,Y 256.068,Z 178.082,A -85,B 0,C 180,E1 -18663.294,E2 -18663.294} C_VEL
LIN {X 0,Y 256.114,Z 178.068,A -85,B 0,C 180,E1 -18667.272,E2 -18667.272} C_VEL
LIN {X 0,Y 256.056,Z 178.09,A -85,B 0,C 180,E1 -18671.205,E2 -18671.205} C_VEL
LIN {X 0,Y 256.063,Z 178.078,A -85,B 0,C 180,E1 -18675.53,E2 -18675.53} C_VEL
LIN {X 0,Y 256.055,Z 178.066,A -85,B 0,C 180,E1 -18678.798,E2 -18678.798} C_VEL
LIN {X 0,Y 256.127,Z 178.078,A -85,B 0,C 180,E1 -18682.868,E2 -18682.868} C_VEL
LIN {X 0,Y 256.067,Z 178.087,A -85,B 0,C 180,E1 -18686.708,E2 -18686.708} C_VEL
LIN {X 0,Y 256.056,Z 178.086,A -85,B 0,C 180,E1 -18690.394,E2 -18690.394} C_VEL
LIN {X 0,Y 256.135,Z 178.076,A -85,B 0,C 180,E1 -18694.889,E2 -18694.889} C_VEL
LIN {X 0,Y 256.165,Z 178.072,A -85,B 0,C 180,E1 -18699.106,E2 -18699.106} C_VEL
LIN {X 0,Y 256.264,Z 178.059,A -85,B 0,C 180,E1 -18703.716,E2 -18703.716} C_VEL
LIN {X 0,Y 256.295,Z 178.056,A -85,B 0,C 180,E1 -18707.329,E2 -18707.329} C_VEL
LIN {X 0,Y 256.437,Z 178.037,A -85,B 0,C 180,E1 -18710.624,E2 -18710.624} C_VEL
LIN {X 0,Y 256.457,Z 178.035,A -85,B 0,C 180,E1 -18713.707,E2 -18713.707} C_VEL
LIN {X 0,Y 256.702,Z 178.004,A -85,B 0,C 180,E1 -18718.432,E2 -18718.432} C_VEL
LIN {X 0,Y 256.7,Z 177.991,A -85,B 0,C 180,E1 -18721.57,E2 -18721.57} C_VEL
LIN {X 0,Y 256.329,Z 178.037,A -85,B 0,C 180,E1 -18725.157,E2 -18725.157} C_VEL
LIN {X 0,Y 255.723,Z 178.123,A -85,B 0,C 180,E1 -18726.471,E2 -18726.471} C_VEL
LIN {X 0,Y 252.86,Z 178.485,A -85,B 0,C 180,E1 -18728.61,E2 -18728.61} C_VEL
LIN {X 0,Y 250.374,Z 178.796,A -85,B 0,C 180,E1 -18730.352,E2 -18730.352} C_VEL
LIN {X 0,Y 249.287,Z 178.93,A -85,B 0,C 180,E1 -18731.704,E2 -18731.704} C_VEL
LIN {X 0,Y 249.19,Z 178.939,A -85,B 0,C 180,E1 -18732.163,E2 -18732.163} C_VEL
LIN {X 0,Y 249.178,Z 178.927,A -85,B 0,C 180,E1 -18736.468,E2 -18736.468} C_VEL
LIN {X 0,Y 249.047,Z 178.963,A -85,B 0,C 180,E1 -18741.522,E2 -18741.522} C_VEL
LIN {X 0,Y 249.051,Z 178.947,A -85,B 0,C 180,E1 -18745.441,E2 -18745.441} C_VEL
LIN {X 0,Y 249.038,Z 178.962,A -85,B 0,C 180,E1 -18748.972,E2 -18748.972} C_VEL
LIN {X 0,Y 249.032,Z 178.961,A -85,B 0,C 180,E1 -18752.426,E2 -18752.426} C_VEL
LIN {X 0,Y 249.031,Z 178.962,A -85,B 0,C 180,E1 -18756.346,E2 -18756.346} C_VEL
LIN {X 0,Y 248.983,Z 178.961,A -85,B 0,C 180,E1 -18760.483,E2 -18760.483} C_VEL
LIN {X 0,Y 248.966,Z 178.967,A -85,B 0,C 180,E1 -18764.889,E2 -18764.889} C_VEL
LIN {X 0,Y 248.981,Z 178.97,A -85,B 0,C 180,E1 -18767.354,E2 -18767.354} C_VEL
LIN {X 0,Y 249.026,Z 178.966,A -85,B 0,C 180,E1 -18772.207,E2 -18772.207} C_VEL
LIN {X 0,Y 249.077,Z 179.057,A -85,B 0,C 180,E1 -18775.067,E2 -18775.067} C_VEL
LIN {X 0,Y 251.285,Z 189.397,A -85,B 0,C 180,E1 -18779.307,E2 -18779.307} C_VEL
LIN {X 0,Y 251.636,Z 191.106,A -85,B 0,C 180,E1 -18779.818,E2 -18779.818} C_VEL
LIN {X 0,Y 258.857,Z 210.744,A -85,B 0,C 180,E1 -18781.23,E2 -18781.23} C_VEL
LIN {X 0,Y 262.599,Z 236.594,A -85,B 0,C 180,E1 -18782.422,E2 -18782.422} C_VEL
LIN {X 0,Y 260.387,Z 298.78,A -85,B 0,C 180,E1 -18784.265,E2 -18784.265} C_VEL
LIN {X 0,Y 259.372,Z 312.192,A -85,B 0,C 180,E1 -18784.951,E2 -18784.951} C_VEL
LIN {X 0,Y 258.131,Z 324.668,A -85,B 0,C 180,E1 -18785.894,E2 -18785.894} C_VEL
LIN {X 0,Y 256.67,Z 335.868,A -85,B 0,C 180,E1 -18787.033,E2 -18787.033} C_VEL
LIN {X 0,Y 255.094,Z 346.224,A -85,B 0,C 180,E1 -18788.376,E2 -18788.376} C_VEL
LIN {X 0,Y 253.39,Z 356.978,A -85,B 0,C 180,E1 -18790.136,E2 -18790.136} C_VEL
LIN {X 0,Y 251.818,Z 366.678,A -85,B 0,C 180,E1 -18792.12,E2 -18792.12} C_VEL
LIN {X 0,Y 250.389,Z 374.595,A -85,B 0,C 180,E1 -18794.116,E2 -18794.116} C_VEL
